Yaskawa INFORM job: A_ROOF_SIDE_0617_2_PAINT_49.JBI

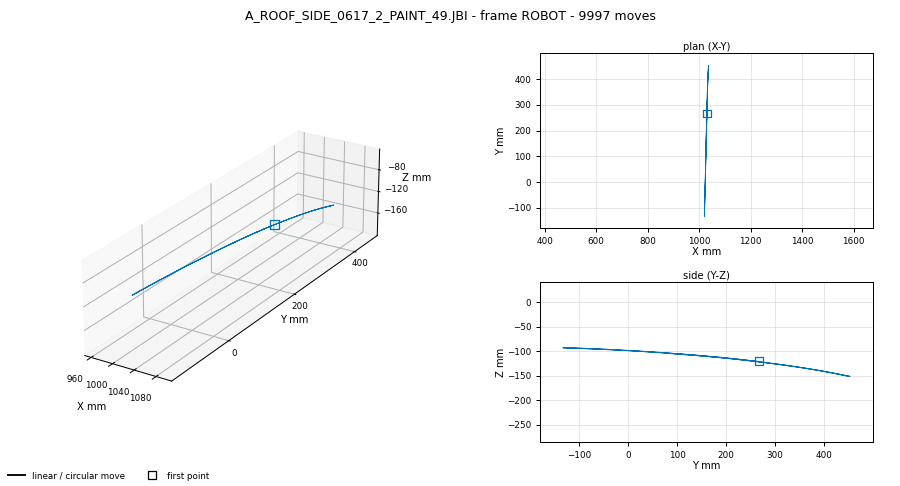
[picture p0: tool path of A_ROOF_SIDE_0617_2_PAINT_49.JBI in frame ROBOT, 9997 of 9997 moves have a stored position in this frame; points joined in program order, loops and branches not executed]
/JOB
//NAME A_ROOF_SIDE_0617_2_PAINT49
//POS
///NPOS 9997,0,0,0,0,0
///TOOL 1
///USER 0
///POSTYPE ROBOT
///RECTAN
///RCONF 1,0,0,0,0,0,0,0,0,0,0,0,0,0,0,0,0,0,0,0,0,0,0,0
C00000=1029.907,266.223,-120.891,170.566,45.689,158.767
C00001=1029.902,265.975,-120.861,170.562,45.690,158.767
C00002=1029.894,265.727,-120.831,170.558,45.691,158.767
C00003=1029.887,265.479,-120.801,170.555,45.691,158.766
C00004=1029.881,265.230,-120.772,170.551,45.692,158.766
C00005=1029.874,264.982,-120.741,170.547,45.693,158.766
C00006=1029.868,264.734,-120.711,170.544,45.694,158.766
C00007=1029.861,264.486,-120.681,170.539,45.695,158.766
C00008=1029.854,264.238,-120.651,170.536,45.696,158.765
C00009=1029.847,263.990,-120.622,170.532,45.697,158.765
C00010=1029.837,263.620,-120.577,170.527,45.697,158.765
C00011=1029.828,263.250,-120.532,170.521,45.699,158.764
C00012=1029.817,262.880,-120.488,170.516,45.700,158.764
C00013=1029.807,262.510,-120.443,170.511,45.701,158.764
C00014=1029.802,262.262,-120.413,170.507,45.702,158.764
C00015=1029.795,262.013,-120.383,170.503,45.703,158.763
C00016=1029.788,261.765,-120.354,170.500,45.704,158.763
C00017=1029.781,261.517,-120.324,170.496,45.705,158.763
C00018=1029.775,261.270,-120.294,170.493,45.705,158.763
C00019=1029.768,261.020,-120.264,170.489,45.706,158.763
C00020=1029.761,260.773,-120.235,170.486,45.708,158.763
C00021=1029.754,260.524,-120.205,170.482,45.709,158.762
C00022=1029.748,260.277,-120.176,170.478,45.710,158.762
C00023=1029.741,260.028,-120.146,170.475,45.710,158.762
C00024=1029.734,259.781,-120.117,170.471,45.711,158.762
C00025=1029.727,259.532,-120.088,170.468,45.713,158.762
C00026=1029.720,259.285,-120.058,170.464,45.714,158.761
C00027=1029.713,259.036,-120.029,170.460,45.715,158.761
C00028=1029.707,258.788,-120.000,170.457,45.715,158.761
C00029=1029.700,258.539,-119.969,170.453,45.717,158.761
C00030=1029.694,258.291,-119.940,170.450,45.718,158.761
C00031=1029.686,258.043,-119.912,170.446,45.719,158.761
C00032=1029.680,257.795,-119.882,170.442,45.720,158.760
C00033=1029.673,257.546,-119.852,170.439,45.721,158.760
C00034=1029.666,257.298,-119.823,170.435,45.722,158.760
C00035=1029.659,257.050,-119.793,170.432,45.723,158.760
C00036=1029.652,256.802,-119.765,170.428,45.724,158.760
C00037=1029.645,256.553,-119.735,170.425,45.725,158.760
C00038=1029.639,256.306,-119.706,170.421,45.726,158.760
C00039=1029.633,256.058,-119.677,170.417,45.727,158.759
C00040=1029.626,255.809,-119.647,170.414,45.728,158.759
C00041=1029.619,255.561,-119.619,170.410,45.729,158.759
C00042=1029.612,255.313,-119.589,170.407,45.730,158.759
C00043=1029.605,255.065,-119.560,170.403,45.731,158.759
C00044=1029.599,254.817,-119.531,170.401,45.732,158.759
C00045=1029.592,254.568,-119.501,170.397,45.733,158.758
C00046=1029.585,254.321,-119.472,170.393,45.734,158.758
C00047=1029.579,254.072,-119.443,170.390,45.735,158.758
C00048=1029.572,253.824,-119.414,170.387,45.736,158.758
C00049=1029.566,253.575,-119.385,170.383,45.737,158.758
C00050=1029.559,253.327,-119.355,170.380,45.739,158.758
C00051=1029.552,253.079,-119.327,170.376,45.739,158.758
C00052=1029.546,252.831,-119.298,170.372,45.740,158.757
C00053=1029.538,252.582,-119.267,170.369,45.742,158.757
C00054=1029.532,252.334,-119.238,170.365,45.743,158.757
C00055=1029.526,252.086,-119.209,170.362,45.743,158.757
C00056=1029.519,251.838,-119.181,170.358,45.745,158.757
C00057=1029.512,251.590,-119.152,170.355,45.746,158.757
C00058=1029.506,251.341,-119.123,170.351,45.747,158.757
C00059=1029.500,251.093,-119.093,170.348,45.748,158.756
C00060=1029.492,250.845,-119.065,170.344,45.749,158.756
C00061=1029.486,250.597,-119.036,170.342,45.750,158.756
C00062=1029.479,250.349,-119.007,170.337,45.751,158.756
C00063=1029.473,250.100,-118.978,170.335,45.753,158.756
C00064=1029.466,249.852,-118.948,170.332,45.753,158.756
C00065=1029.459,249.604,-118.920,170.328,45.754,158.756
C00066=1029.450,249.232,-118.876,170.323,45.756,158.755
C00067=1029.440,248.861,-118.833,170.318,45.758,158.755
C00068=1029.431,248.490,-118.789,170.312,45.760,158.755
C00069=1029.421,248.118,-118.746,170.307,45.761,158.755
C00070=1029.413,247.870,-118.717,170.304,45.762,158.755
C00071=1029.407,247.622,-118.688,170.300,45.764,158.755
C00072=1029.401,247.373,-118.660,170.297,45.764,158.754
C00073=1029.395,247.125,-118.631,170.295,45.766,158.754
C00074=1029.389,246.877,-118.602,170.291,45.767,158.754
C00075=1029.381,246.628,-118.573,170.288,45.768,158.754
C00076=1029.375,246.380,-118.544,170.284,45.769,158.754
C00077=1029.369,246.132,-118.515,170.281,45.770,158.754
C00078=1029.362,245.884,-118.486,170.277,45.771,158.754
C00079=1029.356,245.635,-118.458,170.274,45.773,158.754
C00080=1029.349,245.387,-118.429,170.271,45.774,158.753
C00081=1029.343,245.139,-118.400,170.267,45.774,158.753
C00082=1029.336,244.890,-118.371,170.264,45.776,158.753
C00083=1029.329,244.642,-118.342,170.260,45.777,158.753
C00084=1029.323,244.394,-118.314,170.258,45.778,158.753
C00085=1029.317,244.145,-118.285,170.254,45.780,158.753
C00086=1029.310,243.898,-118.256,170.251,45.780,158.753
C00087=1029.304,243.649,-118.228,170.248,45.782,158.753
C00088=1029.297,243.401,-118.200,170.244,45.783,158.752
C00089=1029.291,243.153,-118.170,170.241,45.784,158.752
C00090=1029.284,242.904,-118.142,170.237,45.786,158.752
C00091=1029.277,242.656,-118.113,170.234,45.786,158.752
C00092=1029.271,242.407,-118.086,170.231,45.788,158.752
C00093=1029.265,242.159,-118.057,170.228,45.789,158.752
C00094=1029.258,241.911,-118.028,170.224,45.790,158.752
C00095=1029.252,241.662,-118.000,170.221,45.792,158.752
C00096=1029.245,241.415,-117.971,170.218,45.793,158.752
C00097=1029.239,241.166,-117.943,170.214,45.794,158.752
C00098=1029.232,240.918,-117.915,170.211,45.795,158.752
C00099=1029.226,240.669,-117.886,170.208,45.797,158.752
C00100=1029.219,240.422,-117.858,170.205,45.798,158.751
C00101=1029.213,240.173,-117.829,170.202,45.799,158.751
C00102=1029.205,239.924,-117.801,170.198,45.801,158.751
C00103=1029.199,239.676,-117.773,170.195,45.802,158.751
C00104=1029.192,239.428,-117.744,170.191,45.803,158.751
C00105=1029.185,239.180,-117.717,170.188,45.804,158.751
C00106=1029.179,238.931,-117.688,170.185,45.806,158.751
C00107=1029.172,238.683,-117.660,170.182,45.807,158.751
C00108=1029.165,238.435,-117.632,170.178,45.809,158.751
C00109=1029.159,238.186,-117.605,170.175,45.810,158.751
C00110=1029.152,237.938,-117.575,170.172,45.811,158.751
C00111=1029.146,237.689,-117.548,170.169,45.813,158.751
C00112=1029.139,237.441,-117.520,170.166,45.814,158.751
C00113=1029.132,237.193,-117.492,170.162,45.816,158.751
C00114=1029.126,236.944,-117.463,170.159,45.817,158.751
C00115=1029.119,236.696,-117.436,170.157,45.818,158.751
C00116=1029.113,236.448,-117.408,170.153,45.820,158.750
C00117=1029.106,236.200,-117.379,170.150,45.821,158.750
C00118=1029.099,235.951,-117.352,170.146,45.822,158.750
C00119=1029.092,235.703,-117.324,170.143,45.824,158.750
C00120=1029.086,235.454,-117.296,170.139,45.825,158.750
C00121=1029.080,235.206,-117.268,170.137,45.827,158.750
C00122=1029.070,234.829,-117.225,170.132,45.829,158.750
C00123=1029.059,234.451,-117.182,170.127,45.831,158.750
C00124=1029.049,234.073,-117.140,170.123,45.833,158.750
C00125=1029.039,233.696,-117.098,170.117,45.836,158.750
C00126=1029.033,233.448,-117.070,170.114,45.837,158.750
C00127=1029.026,233.199,-117.042,170.111,45.838,158.750
C00128=1029.019,232.951,-117.014,170.107,45.839,158.750
C00129=1029.013,232.702,-116.987,170.105,45.841,158.750
C00130=1029.006,232.454,-116.959,170.102,45.842,158.750
C00131=1029.000,232.205,-116.931,170.098,45.844,158.750
C00132=1028.993,231.957,-116.903,170.095,45.845,158.750
C00133=1028.987,231.708,-116.875,170.092,45.847,158.749
C00134=1028.981,231.461,-116.848,170.089,45.848,158.749
C00135=1028.974,231.212,-116.820,170.086,45.849,158.749
C00136=1028.967,230.964,-116.792,170.082,45.851,158.749
C00137=1028.960,230.715,-116.765,170.080,45.852,158.749
C00138=1028.954,230.467,-116.737,170.077,45.854,158.749
C00139=1028.947,230.218,-116.709,170.073,45.855,158.749
C00140=1028.940,229.970,-116.681,170.070,45.857,158.749
C00141=1028.934,229.722,-116.654,170.066,45.858,158.749
C00142=1028.927,229.473,-116.626,170.064,45.860,158.749
C00143=1028.921,229.225,-116.599,170.061,45.861,158.749
C00144=1028.914,228.977,-116.571,170.057,45.863,158.749
C00145=1028.908,228.728,-116.543,170.055,45.865,158.749
C00146=1028.901,228.480,-116.515,170.052,45.866,158.749
C00147=1028.894,228.232,-116.488,170.048,45.868,158.749
C00148=1028.888,227.983,-116.461,170.045,45.869,158.749
C00149=1028.881,227.734,-116.433,170.043,45.870,158.749
C00150=1028.875,227.486,-116.406,170.039,45.872,158.749
C00151=1028.868,227.238,-116.378,170.036,45.873,158.749
C00152=1028.862,226.989,-116.350,170.032,45.875,158.749
C00153=1028.855,226.741,-116.324,170.030,45.876,158.749
C00154=1028.848,226.492,-116.296,170.027,45.878,158.749
C00155=1028.841,226.244,-116.268,170.023,45.880,158.749
C00156=1028.835,225.996,-116.241,170.021,45.881,158.749
C00157=1028.828,225.747,-116.214,170.018,45.883,158.749
C00158=1028.821,225.499,-116.187,170.014,45.885,158.749
C00159=1028.815,225.250,-116.159,170.012,45.886,158.749
C00160=1028.808,225.001,-116.132,170.009,45.888,158.749
C00161=1028.802,224.754,-116.105,170.005,45.889,158.749
C00162=1028.795,224.506,-116.078,170.002,45.891,158.749
C00163=1028.788,224.256,-116.050,169.999,45.893,158.749
C00164=1028.782,224.008,-116.023,169.996,45.894,158.749
C00165=1028.774,223.760,-115.996,169.993,45.896,158.749
C00166=1028.769,223.512,-115.969,169.989,45.897,158.749
C00167=1028.762,223.263,-115.941,169.987,45.899,158.749
C00168=1028.756,223.014,-115.914,169.984,45.901,158.749
C00169=1028.748,222.766,-115.887,169.980,45.902,158.749
C00170=1028.742,222.518,-115.860,169.978,45.904,158.749
C00171=1028.736,222.269,-115.833,169.975,45.906,158.749
C00172=1028.728,222.021,-115.806,169.971,45.907,158.749
C00173=1028.722,221.772,-115.779,169.969,45.909,158.749
C00174=1028.716,221.524,-115.751,169.966,45.910,158.749
C00175=1028.709,221.275,-115.724,169.962,45.912,158.749
C00176=1028.702,221.027,-115.697,169.960,45.914,158.749
C00177=1028.696,220.778,-115.670,169.957,45.915,158.749
C00178=1028.686,220.394,-115.628,169.952,45.918,158.749
C00179=1028.675,220.008,-115.586,169.948,45.920,158.749
C00180=1028.665,219.623,-115.544,169.942,45.923,158.749
C00181=1028.656,219.237,-115.502,169.938,45.925,158.749
C00182=1028.648,218.989,-115.475,169.935,45.927,158.749
C00183=1028.643,218.741,-115.448,169.932,45.929,158.749
C00184=1028.635,218.492,-115.422,169.929,45.930,158.749
C00185=1028.628,218.244,-115.394,169.926,45.932,158.749
C00186=1028.622,217.995,-115.367,169.923,45.934,158.749
C00187=1028.615,217.747,-115.341,169.920,45.936,158.749
C00188=1028.608,217.499,-115.314,169.917,45.937,158.749
C00189=1028.601,217.250,-115.287,169.915,45.939,158.750
C00190=1028.596,217.001,-115.261,169.911,45.941,158.750
C00191=1028.588,216.753,-115.233,169.908,45.943,158.750
C00192=1028.582,216.504,-115.206,169.906,45.944,158.750
C00193=1028.575,216.256,-115.180,169.902,45.946,158.750
C00194=1028.569,216.007,-115.153,169.899,45.948,158.750
C00195=1028.561,215.759,-115.126,169.897,45.949,158.750
C00196=1028.555,215.511,-115.100,169.893,45.952,158.750
C00197=1028.549,215.262,-115.073,169.890,45.953,158.750
C00198=1028.542,215.014,-115.047,169.888,45.955,158.750
C00199=1028.536,214.765,-115.020,169.884,45.957,158.750
C00200=1028.528,214.517,-114.993,169.882,45.959,158.750
C00201=1028.523,214.268,-114.966,169.879,45.960,158.750
C00202=1028.515,214.020,-114.940,169.876,45.962,158.750
C00203=1028.508,213.771,-114.913,169.873,45.964,158.750
C00204=1028.503,213.522,-114.887,169.870,45.966,158.750
C00205=1028.495,213.274,-114.860,169.867,45.967,158.750
C00206=1028.489,213.026,-114.833,169.864,45.969,158.750
C00207=1028.482,212.777,-114.807,169.861,45.971,158.750
C00208=1028.476,212.529,-114.780,169.859,45.973,158.750
C00209=1028.469,212.280,-114.754,169.856,45.974,158.750
C00210=1028.463,212.031,-114.727,169.852,45.976,158.751
C00211=1028.456,211.783,-114.700,169.850,45.978,158.750
C00212=1028.449,211.534,-114.674,169.847,45.980,158.751
C00213=1028.444,211.286,-114.647,169.843,45.981,158.751
C00214=1028.436,211.038,-114.620,169.841,45.983,158.751
C00215=1028.430,210.789,-114.594,169.838,45.985,158.751
C00216=1028.423,210.541,-114.567,169.836,45.987,158.751
C00217=1028.417,210.293,-114.541,169.832,45.988,158.751
C00218=1028.410,210.044,-114.515,169.829,45.990,158.751
C00219=1028.403,209.795,-114.488,169.827,45.993,158.751
C00220=1028.397,209.547,-114.462,169.823,45.994,158.751
C00221=1028.390,209.298,-114.435,169.821,45.996,158.751
C00222=1028.383,209.050,-114.409,169.818,45.998,158.751
C00223=1028.377,208.800,-114.383,169.815,46.000,158.751
C00224=1028.371,208.552,-114.357,169.812,46.002,158.751
C00225=1028.363,208.303,-114.330,169.809,46.003,158.751
C00226=1028.357,208.055,-114.304,169.807,46.005,158.751
C00227=1028.351,207.806,-114.277,169.803,46.008,158.752
C00228=1028.344,207.558,-114.251,169.801,46.010,158.752
C00229=1028.337,207.309,-114.225,169.798,46.011,158.752
C00230=1028.330,207.061,-114.199,169.795,46.013,158.752
C00231=1028.323,206.813,-114.172,169.792,46.015,158.752
C00232=1028.317,206.564,-114.147,169.789,46.017,158.752
C00233=1028.311,206.315,-114.120,169.787,46.019,158.752
C00234=1028.300,205.936,-114.080,169.782,46.022,158.752
C00235=1028.290,205.556,-114.040,169.778,46.024,158.752
C00236=1028.280,205.176,-114.001,169.774,46.027,158.752
C00237=1028.269,204.795,-113.961,169.769,46.031,158.753
C00238=1028.244,203.751,-113.857,169.396,45.927,158.689
C00239=1028.238,203.502,-113.832,169.392,45.930,158.689
C00240=1028.233,203.253,-113.808,169.388,45.932,158.689
C00241=1028.227,203.005,-113.783,169.384,45.936,158.690
C00242=1028.220,202.756,-113.759,169.380,45.938,158.690
C00243=1028.215,202.508,-113.734,169.376,45.941,158.690
C00244=1028.209,202.258,-113.709,169.372,45.943,158.690
C00245=1028.203,202.009,-113.684,169.369,45.946,158.690
C00246=1028.197,201.761,-113.659,169.365,45.949,158.690
C00247=1028.191,201.512,-113.635,169.361,45.952,158.690
C00248=1028.185,201.264,-113.611,169.357,45.954,158.690
C00249=1028.179,201.015,-113.586,169.354,45.957,158.691
C00250=1028.174,200.766,-113.562,169.349,45.960,158.691
C00251=1028.168,200.517,-113.537,169.346,45.963,158.691
C00252=1028.162,200.268,-113.512,169.342,45.965,158.691
C00253=1028.156,200.020,-113.488,169.338,45.968,158.691
C00254=1028.150,199.771,-113.463,169.335,45.971,158.691
C00255=1028.144,199.523,-113.440,169.331,45.974,158.692
C00256=1028.138,199.273,-113.415,169.327,45.976,158.692
C00257=1028.132,199.025,-113.391,169.323,45.980,158.692
C00258=1028.126,198.776,-113.367,169.320,45.982,158.692
C00259=1028.119,198.527,-113.343,169.315,45.985,158.692
C00260=1028.113,198.278,-113.319,169.312,45.988,158.692
C00261=1028.107,198.030,-113.294,169.308,45.991,158.692
C00262=1028.101,197.782,-113.270,169.304,45.994,158.693
C00263=1028.095,197.532,-113.245,169.301,45.996,158.693
C00264=1028.089,197.284,-113.222,169.297,45.999,158.693
C00265=1028.083,197.035,-113.197,169.293,46.002,158.693
C00266=1028.077,196.786,-113.173,169.289,46.006,158.693
C00267=1028.071,196.537,-113.149,169.286,46.008,158.693
C00268=1028.065,196.289,-113.125,169.282,46.011,158.694
C00269=1028.059,196.040,-113.101,169.278,46.014,158.694
C00270=1028.053,195.791,-113.077,169.275,46.017,158.694
C00271=1028.047,195.542,-113.053,169.271,46.020,158.694
C00272=1028.041,195.294,-113.029,169.267,46.022,158.694
C00273=1028.035,195.045,-113.005,169.264,46.025,158.695
C00274=1028.030,194.795,-112.981,169.260,46.028,158.695
C00275=1028.024,194.547,-112.957,169.256,46.031,158.695
C00276=1028.018,194.298,-112.933,169.252,46.035,158.695
C00277=1028.012,194.050,-112.909,169.249,46.037,158.695
C00278=1028.006,193.800,-112.885,169.245,46.040,158.695
C00279=1028.000,193.552,-112.861,169.241,46.043,158.696
C00280=1027.993,193.303,-112.837,169.238,46.046,158.696
C00281=1027.988,193.055,-112.813,169.235,46.049,158.696
C00282=1027.982,192.806,-112.789,169.230,46.051,158.696
C00283=1027.976,192.556,-112.765,169.227,46.054,158.696
C00284=1027.970,192.308,-112.741,169.224,46.057,158.697
C00285=1027.965,192.059,-112.717,169.219,46.060,158.697
C00286=1027.958,191.810,-112.693,169.216,46.063,158.697
C00287=1027.952,191.562,-112.669,169.213,46.066,158.697
C00288=1027.947,191.312,-112.645,169.208,46.069,158.697
C00289=1027.941,191.064,-112.622,169.205,46.072,158.697
C00290=1027.935,190.815,-112.598,169.202,46.075,158.698
C00291=1027.929,190.566,-112.574,169.198,46.078,158.698
C00292=1027.924,190.317,-112.550,169.194,46.081,158.698
C00293=1027.918,190.069,-112.526,169.191,46.083,158.698
C00294=1027.912,189.821,-112.503,169.187,46.086,158.698
C00295=1027.906,189.571,-112.478,169.183,46.089,158.699
C00296=1027.900,189.323,-112.455,169.180,46.092,158.699
C00297=1027.895,189.074,-112.431,169.177,46.095,158.699
C00298=1027.888,188.825,-112.407,169.173,46.098,158.699
C00299=1027.882,188.542,-112.379,169.169,46.101,158.699
C00300=1027.875,188.259,-112.353,169.165,46.104,158.700
C00301=1027.869,187.976,-112.326,169.161,46.108,158.700
C00302=1027.862,187.693,-112.299,169.157,46.111,158.700
C00303=1027.857,187.444,-112.275,169.154,46.114,158.700
C00304=1027.851,187.196,-112.252,169.149,46.117,158.700
C00305=1027.844,186.947,-112.228,169.146,46.120,158.701
C00306=1027.839,186.697,-112.204,169.143,46.123,158.701
C00307=1027.833,186.449,-112.181,169.140,46.126,158.701
C00308=1027.828,186.200,-112.157,169.135,46.129,158.701
C00309=1027.822,185.952,-112.133,169.132,46.132,158.701
C00310=1027.815,185.703,-112.109,169.129,46.135,158.702
C00311=1027.810,185.453,-112.086,169.125,46.137,158.702
C00312=1027.804,185.205,-112.062,169.122,46.140,158.702
C00313=1027.799,184.956,-112.039,169.118,46.143,158.702
C00314=1027.793,184.708,-112.015,169.115,46.146,158.702
C00315=1027.787,184.459,-111.992,169.111,46.149,158.703
C00316=1027.782,184.209,-111.967,169.108,46.152,158.703
C00317=1027.776,183.961,-111.944,169.105,46.155,158.703
C00318=1027.771,183.712,-111.920,169.101,46.158,158.703
C00319=1027.765,183.463,-111.897,169.097,46.161,158.703
C00320=1027.759,183.215,-111.874,169.094,46.164,158.703
C00321=1027.753,182.965,-111.850,169.091,46.166,158.704
C00322=1027.747,182.716,-111.827,169.087,46.169,158.704
C00323=1027.741,182.468,-111.803,169.083,46.173,158.704
C00324=1027.736,182.219,-111.780,169.080,46.176,158.705
C00325=1027.729,181.969,-111.757,169.077,46.179,158.705
C00326=1027.723,181.721,-111.734,169.073,46.182,158.705
C00327=1027.717,181.472,-111.711,169.070,46.185,158.705
C00328=1027.711,181.223,-111.689,169.066,46.188,158.705
C00329=1027.705,180.975,-111.665,169.063,46.192,158.706
C00330=1027.700,180.726,-111.642,169.059,46.195,158.706
C00331=1027.693,180.476,-111.619,169.056,46.198,158.706
C00332=1027.687,180.227,-111.596,169.053,46.201,158.706
C00333=1027.681,179.979,-111.573,169.048,46.204,158.707
C00334=1027.675,179.730,-111.550,169.045,46.208,158.707
C00335=1027.669,179.481,-111.528,169.042,46.211,158.707
C00336=1027.663,179.232,-111.505,169.039,46.214,158.707
C00337=1027.657,178.983,-111.481,169.035,46.217,158.708
C00338=1027.651,178.734,-111.458,169.032,46.221,158.708
C00339=1027.645,178.485,-111.435,169.029,46.224,158.708
C00340=1027.639,178.237,-111.413,169.025,46.227,158.708
C00341=1027.633,177.988,-111.390,169.022,46.230,158.709
C00342=1027.627,177.739,-111.367,169.018,46.233,158.709
C00343=1027.621,177.490,-111.344,169.015,46.236,158.709
C00344=1027.615,177.242,-111.322,169.012,46.239,158.709
C00345=1027.609,176.992,-111.298,169.009,46.242,158.710
C00346=1027.603,176.743,-111.275,169.004,46.245,158.710
C00347=1027.597,176.494,-111.252,169.001,46.249,158.710
C00348=1027.591,176.246,-111.230,168.998,46.252,158.710
C00349=1027.585,175.997,-111.207,168.995,46.255,158.711
C00350=1027.579,175.748,-111.184,168.992,46.258,158.711
C00351=1027.573,175.499,-111.161,168.988,46.262,158.711
C00352=1027.567,175.250,-111.139,168.984,46.265,158.711
C00353=1027.561,175.001,-111.116,168.981,46.268,158.712
C00354=1027.556,174.753,-111.093,168.978,46.271,158.712
C00355=1027.550,174.504,-111.070,168.975,46.274,158.712
C00356=1027.544,174.254,-111.048,168.972,46.277,158.712
C00357=1027.538,174.006,-111.025,168.968,46.281,158.713
C00358=1027.532,173.757,-111.003,168.964,46.284,158.713
C00359=1027.526,173.508,-110.980,168.961,46.287,158.713
C00360=1027.520,173.259,-110.957,168.958,46.290,158.714
C00361=1027.514,173.010,-110.934,168.955,46.293,158.714
C00362=1027.509,172.761,-110.911,168.952,46.296,158.714
C00363=1027.502,172.478,-110.886,168.948,46.300,158.714
C00364=1027.495,172.194,-110.860,168.944,46.304,158.715
C00365=1027.488,171.911,-110.834,168.940,46.308,158.715
C00366=1027.482,171.627,-110.808,168.937,46.311,158.715
C00367=1027.476,171.378,-110.786,168.934,46.314,158.716
C00368=1027.470,171.129,-110.763,168.930,46.317,158.716
C00369=1027.464,170.881,-110.740,168.926,46.320,158.716
C00370=1027.459,170.631,-110.718,168.923,46.323,158.716
C00371=1027.452,170.382,-110.695,168.920,46.327,158.717
C00372=1027.447,170.134,-110.673,168.917,46.330,158.717
C00373=1027.441,169.885,-110.650,168.914,46.333,158.717
C00374=1027.435,169.635,-110.627,168.910,46.336,158.717
C00375=1027.430,169.387,-110.605,168.907,46.340,158.718
C00376=1027.424,169.138,-110.582,168.904,46.343,158.718
C00377=1027.418,168.889,-110.559,168.901,46.346,158.718
C00378=1027.412,168.640,-110.538,168.898,46.349,158.718
C00379=1027.406,168.391,-110.515,168.894,46.352,158.719
C00380=1027.401,168.142,-110.492,168.891,46.355,158.719
C00381=1027.395,167.893,-110.470,168.887,46.358,158.719
C00382=1027.389,167.644,-110.447,168.884,46.362,158.719
C00383=1027.383,167.396,-110.425,168.881,46.365,158.720
C00384=1027.378,167.147,-110.403,168.878,46.368,158.720
C00385=1027.372,166.898,-110.380,168.875,46.371,158.720
C00386=1027.366,166.649,-110.357,168.872,46.375,158.720
C00387=1027.360,166.400,-110.335,168.869,46.378,158.721
C00388=1027.355,166.151,-110.312,168.865,46.381,158.721
C00389=1027.349,165.902,-110.291,168.862,46.384,158.721
C00390=1027.343,165.653,-110.268,168.859,46.387,158.722
C00391=1027.338,165.404,-110.245,168.856,46.390,158.722
C00392=1027.332,165.155,-110.223,168.853,46.393,158.722
C00393=1027.326,164.906,-110.200,168.850,46.397,158.722
C00394=1027.320,164.657,-110.178,168.847,46.400,158.723
C00395=1027.315,164.409,-110.156,168.843,46.403,158.723
C00396=1027.309,164.160,-110.133,168.840,46.406,158.723
C00397=1027.303,163.911,-110.111,168.837,46.409,158.723
C00398=1027.298,163.662,-110.088,168.834,46.412,158.724
C00399=1027.292,163.413,-110.067,168.831,46.415,158.724
C00400=1027.286,163.164,-110.044,168.827,46.418,158.724
C00401=1027.281,162.915,-110.022,168.825,46.422,158.724
C00402=1027.275,162.666,-109.999,168.821,46.425,158.725
C00403=1027.270,162.417,-109.977,168.818,46.428,158.725
C00404=1027.264,162.168,-109.954,168.815,46.432,158.725
C00405=1027.258,161.919,-109.932,168.812,46.435,158.726
C00406=1027.252,161.670,-109.910,168.809,46.438,158.726
C00407=1027.247,161.422,-109.888,168.805,46.441,158.726
C00408=1027.242,161.172,-109.866,168.803,46.444,158.726
C00409=1027.235,160.923,-109.843,168.799,46.447,158.727
C00410=1027.230,160.675,-109.821,168.796,46.450,158.727
C00411=1027.225,160.426,-109.799,168.793,46.453,158.727
C00412=1027.219,160.176,-109.776,168.790,46.457,158.727
C00413=1027.213,159.928,-109.754,168.787,46.460,158.728
C00414=1027.208,159.679,-109.732,168.784,46.463,158.728
C00415=1027.203,159.429,-109.710,168.781,46.467,158.728
C00416=1027.196,159.181,-109.688,168.777,46.470,158.728
C00417=1027.191,158.932,-109.666,168.774,46.473,158.729
C00418=1027.184,158.683,-109.645,168.771,46.476,158.729
C00419=1027.179,158.433,-109.622,168.768,46.480,158.729
C00420=1027.173,158.184,-109.601,168.765,46.483,158.730
C00421=1027.167,157.936,-109.579,168.762,46.486,158.730
C00422=1027.161,157.687,-109.557,168.759,46.489,158.730
C00423=1027.155,157.438,-109.535,168.756,46.493,158.731
C00424=1027.150,157.189,-109.514,168.753,46.496,158.731
C00425=1027.144,156.940,-109.492,168.750,46.500,158.731
C00426=1027.137,156.691,-109.470,168.747,46.503,158.731
C00427=1027.131,156.407,-109.445,168.743,46.507,158.732
C00428=1027.124,156.124,-109.420,168.740,46.510,158.732
C00429=1027.118,155.839,-109.396,168.736,46.514,158.732
C00430=1027.111,155.556,-109.371,168.733,46.518,158.733
C00431=1027.106,155.306,-109.349,168.730,46.522,158.733
C00432=1027.100,155.057,-109.327,168.727,46.525,158.733
C00433=1027.094,154.809,-109.306,168.724,46.528,158.734
C00434=1027.088,154.559,-109.284,168.721,46.531,158.734
C00435=1027.082,154.310,-109.262,168.718,46.535,158.734
C00436=1027.077,154.061,-109.241,168.714,46.538,158.735
C00437=1027.071,153.812,-109.219,168.711,46.542,158.735
C00438=1027.065,153.563,-109.197,168.708,46.545,158.735
C00439=1027.059,153.314,-109.176,168.705,46.548,158.736
C00440=1027.054,153.065,-109.154,168.702,46.551,158.736
C00441=1027.047,152.816,-109.132,168.699,46.555,158.736
C00442=1027.042,152.567,-109.111,168.696,46.558,158.736
C00443=1027.036,152.318,-109.089,168.693,46.562,158.737
C00444=1027.030,152.069,-109.068,168.690,46.565,158.737
C00445=1027.024,151.820,-109.047,168.687,46.568,158.737
C00446=1027.018,151.571,-109.025,168.684,46.572,158.738
C00447=1027.012,151.323,-109.004,168.681,46.575,158.738
C00448=1027.006,151.073,-108.982,168.678,46.579,158.738
C00449=1027.000,150.825,-108.961,168.675,46.582,158.739
C00450=1026.994,150.576,-108.939,168.672,46.585,158.739
C00451=1026.989,150.325,-108.918,168.668,46.588,158.739
C00452=1026.984,150.077,-108.896,168.666,46.592,158.740
C00453=1026.977,149.828,-108.875,168.663,46.596,158.740
C00454=1026.972,149.579,-108.853,168.659,46.599,158.740
C00455=1026.966,149.330,-108.832,168.657,46.602,158.741
C00456=1026.960,149.082,-108.810,168.654,46.605,158.741
C00457=1026.954,148.832,-108.789,168.651,46.609,158.741
C00458=1026.948,148.583,-108.768,168.648,46.612,158.741
C00459=1026.943,148.334,-108.747,168.645,46.615,158.742
C00460=1026.936,148.085,-108.725,168.642,46.619,158.742
C00461=1026.931,147.836,-108.704,168.639,46.622,158.742
C00462=1026.925,147.587,-108.682,168.636,46.626,158.743
C00463=1026.919,147.338,-108.662,168.633,46.629,158.743
C00464=1026.913,147.089,-108.640,168.630,46.632,158.743
C00465=1026.908,146.840,-108.619,168.627,46.636,158.744
C00466=1026.902,146.590,-108.598,168.624,46.639,158.744
C00467=1026.896,146.342,-108.576,168.621,46.643,158.744
C00468=1026.890,146.093,-108.555,168.618,46.646,158.745
C00469=1026.885,145.844,-108.534,168.616,46.649,158.745
C00470=1026.879,145.594,-108.513,168.613,46.653,158.745
C00471=1026.872,145.346,-108.492,168.610,46.657,158.746
C00472=1026.867,145.096,-108.471,168.607,46.660,158.746
C00473=1026.861,144.848,-108.450,168.604,46.663,158.746
C00474=1026.855,144.599,-108.428,168.601,46.667,158.747
C00475=1026.850,144.350,-108.408,168.598,46.670,158.747
C00476=1026.843,144.101,-108.387,168.595,46.674,158.747
C00477=1026.837,143.852,-108.366,168.592,46.677,158.748
C00478=1026.831,143.602,-108.344,168.589,46.680,158.748
C00479=1026.826,143.354,-108.323,168.586,46.684,158.748
C00480=1026.820,143.104,-108.302,168.583,46.688,158.749
C00481=1026.814,142.856,-108.281,168.580,46.691,158.749
C00482=1026.808,142.606,-108.261,168.577,46.694,158.749
C00483=1026.802,142.358,-108.239,168.575,46.698,158.750
C00484=1026.796,142.108,-108.218,168.572,46.701,158.750
C00485=1026.791,141.859,-108.197,168.569,46.705,158.750
C00486=1026.785,141.609,-108.176,168.566,46.708,158.751
C00487=1026.779,141.361,-108.156,168.563,46.711,158.751
C00488=1026.773,141.112,-108.135,168.560,46.715,158.751
C00489=1026.767,140.863,-108.113,168.557,46.719,158.752
C00490=1026.762,140.614,-108.093,168.553,46.722,158.752
C00491=1026.755,140.330,-108.069,168.551,46.726,158.752
C00492=1026.748,140.046,-108.045,168.547,46.730,158.753
C00493=1026.742,139.762,-108.021,168.544,46.734,158.753
C00494=1026.735,139.477,-107.997,168.541,46.737,158.753
C00495=1026.729,139.228,-107.976,168.538,46.741,158.754
C00496=1026.724,138.979,-107.955,168.535,46.745,158.754
C00497=1026.718,138.730,-107.935,168.532,46.748,158.754
C00498=1026.712,138.481,-107.914,168.529,46.752,158.755
C00499=1026.706,138.231,-107.893,168.526,46.755,158.755
C00500=1026.700,137.983,-107.872,168.523,46.758,158.755
C00501=1026.694,137.733,-107.852,168.521,46.762,158.756
C00502=1026.689,137.484,-107.831,168.518,46.765,158.756
C00503=1026.682,137.235,-107.810,168.515,46.769,158.757
C00504=1026.677,136.986,-107.789,168.512,46.772,158.757
C00505=1026.670,136.737,-107.769,168.509,46.776,158.757
C00506=1026.665,136.488,-107.748,168.506,46.780,158.758
C00507=1026.660,136.239,-107.727,168.503,46.783,158.758
C00508=1026.653,135.990,-107.707,168.500,46.786,158.758
C00509=1026.647,135.741,-107.686,168.497,46.790,158.758
C00510=1026.641,135.492,-107.666,168.495,46.793,158.759
C00511=1026.635,135.242,-107.645,168.492,46.797,158.759
C00512=1026.629,134.994,-107.625,168.489,46.800,158.760
C00513=1026.624,134.744,-107.604,168.486,46.804,158.760
C00514=1026.618,134.495,-107.583,168.483,46.808,158.760
C00515=1026.612,134.246,-107.563,168.480,46.811,158.761
C00516=1026.607,133.997,-107.542,168.477,46.814,158.761
C00517=1026.600,133.748,-107.522,168.475,46.818,158.761
C00518=1026.595,133.499,-107.501,168.472,46.821,158.762
C00519=1026.589,133.251,-107.481,168.469,46.825,158.762
C00520=1026.583,133.001,-107.460,168.466,46.828,158.762
C00521=1026.577,132.752,-107.440,168.463,46.832,158.763
C00522=1026.572,132.503,-107.419,168.460,46.836,158.763
C00523=1026.565,132.253,-107.399,168.458,46.839,158.763
C00524=1026.560,132.004,-107.378,168.456,46.843,158.764
C00525=1026.553,131.756,-107.358,168.452,46.846,158.764
C00526=1026.548,131.507,-107.337,168.450,46.849,158.764
C00527=1026.542,131.257,-107.317,168.447,46.853,158.765
C00528=1026.536,131.008,-107.296,168.443,46.856,158.765
C00529=1026.530,130.759,-107.276,168.442,46.860,158.765
C00530=1026.525,130.510,-107.256,168.439,46.863,158.766
C00531=1026.518,130.261,-107.235,168.436,46.867,158.766
C00532=1026.513,130.012,-107.215,168.433,46.871,158.767
C00533=1026.507,129.763,-107.195,168.430,46.874,158.767
C00534=1026.501,129.513,-107.174,168.427,46.878,158.767
C00535=1026.495,129.264,-107.155,168.424,46.881,158.767
C00536=1026.489,129.015,-107.134,168.421,46.885,158.768
C00537=1026.483,128.767,-107.114,168.419,46.888,158.768
C00538=1026.477,128.517,-107.094,168.416,46.892,158.769
C00539=1026.471,128.268,-107.074,168.413,46.896,158.769
C00540=1026.465,128.019,-107.054,168.410,46.900,158.769
C00541=1026.459,127.769,-107.034,168.407,46.903,158.770
C00542=1026.453,127.520,-107.014,168.404,46.907,158.770
C00543=1026.447,127.271,-106.994,168.402,46.911,158.771
C00544=1026.441,127.022,-106.974,168.399,46.914,158.771
C00545=1026.435,126.773,-106.953,168.397,46.918,158.771
C00546=1026.429,126.524,-106.933,168.394,46.921,158.772
C00547=1026.423,126.275,-106.913,168.391,46.925,158.772
C00548=1026.417,126.026,-106.893,168.388,46.928,158.772
C00549=1026.412,125.777,-106.874,168.385,46.932,158.773
C00550=1026.405,125.527,-106.853,168.382,46.936,158.773
C00551=1026.399,125.278,-106.833,168.380,46.939,158.773
C00552=1026.394,125.029,-106.813,168.377,46.943,158.774
C00553=1026.388,124.781,-106.793,168.374,46.947,158.774
C00554=1026.382,124.531,-106.774,168.371,46.950,158.775
C00555=1026.375,124.247,-106.751,168.368,46.954,158.775
C00556=1026.369,123.962,-106.728,168.364,46.958,158.775
C00557=1026.362,123.678,-106.705,168.362,46.962,158.776
C00558=1026.354,123.393,-106.682,168.359,46.966,158.776
C00559=1026.349,123.144,-106.662,168.356,46.970,158.777
C00560=1026.343,122.895,-106.642,168.353,46.974,158.777
C00561=1026.337,122.647,-106.622,168.350,46.977,158.777
C00562=1026.331,122.397,-106.603,168.347,46.981,158.778
C00563=1026.325,122.148,-106.583,168.345,46.985,158.778
C00564=1026.319,121.900,-106.563,168.342,46.988,158.778
C00565=1026.314,121.650,-106.542,168.339,46.991,158.779
C00566=1026.308,121.400,-106.522,168.336,46.995,158.779
C00567=1026.302,121.151,-106.502,168.334,46.999,158.779
C00568=1026.296,120.903,-106.483,168.332,47.002,158.780
C00569=1026.290,120.653,-106.463,168.329,47.006,158.780
C00570=1026.284,120.404,-106.443,168.326,47.010,158.781
C00571=1026.279,120.155,-106.423,168.323,47.013,158.781
C00572=1026.273,119.906,-106.404,168.320,47.016,158.781
C00573=1026.267,119.656,-106.383,168.318,47.020,158.782
C00574=1026.261,119.408,-106.363,168.315,47.024,158.782
C00575=1026.255,119.158,-106.344,168.312,47.027,158.782
C00576=1026.249,118.909,-106.324,168.309,47.031,158.783
C00577=1026.244,118.660,-106.303,168.307,47.034,158.783
C00578=1026.238,118.411,-106.284,168.304,47.038,158.783
C00579=1026.232,118.162,-106.264,168.301,47.041,158.784
C00580=1026.226,117.913,-106.244,168.298,47.045,158.784
C00581=1026.220,117.664,-106.225,168.296,47.049,158.785
C00582=1026.214,117.415,-106.205,168.293,47.052,158.785
C00583=1026.209,117.165,-106.186,168.290,47.055,158.785
C00584=1026.203,116.916,-106.165,168.288,47.059,158.785
C00585=1026.197,116.667,-106.145,168.286,47.063,158.786
C00586=1026.192,116.418,-106.126,168.283,47.066,158.786
C00587=1026.186,116.169,-106.106,168.280,47.069,158.786
C00588=1026.180,115.920,-106.087,168.277,47.073,158.787
C00589=1026.174,115.670,-106.067,168.275,47.077,158.787
C00590=1026.169,115.421,-106.047,168.272,47.080,158.788
C00591=1026.163,115.172,-106.027,168.269,47.084,158.788
C00592=1026.157,114.922,-106.008,168.266,47.087,158.788
C00593=1026.151,114.673,-105.988,168.264,47.091,158.789
C00594=1026.145,114.425,-105.968,168.261,47.094,158.789
C00595=1026.139,114.175,-105.948,168.258,47.098,158.789
C00596=1026.133,113.926,-105.928,168.256,47.102,158.790
C00597=1026.128,113.677,-105.909,168.253,47.105,158.790
C00598=1026.122,113.428,-105.889,168.250,47.108,158.790
C00599=1026.117,113.178,-105.869,168.247,47.112,158.791
C00600=1026.111,112.929,-105.850,168.245,47.116,158.791
C00601=1026.105,112.680,-105.830,168.242,47.119,158.791
C00602=1026.099,112.431,-105.811,168.239,47.122,158.792
C00603=1026.093,112.182,-105.791,168.236,47.126,158.792
C00604=1026.088,111.932,-105.772,168.235,47.130,158.793
C00605=1026.082,111.683,-105.753,168.232,47.133,158.793
C00606=1026.075,111.435,-105.733,168.229,47.137,158.793
C00607=1026.069,111.185,-105.714,168.226,47.141,158.794
C00608=1026.064,110.936,-105.695,168.224,47.144,158.794
C00609=1026.058,110.687,-105.675,168.221,47.148,158.794
C00610=1026.052,110.437,-105.655,168.218,47.152,158.795
C00611=1026.046,110.188,-105.636,168.215,47.156,158.795
C00612=1026.041,109.939,-105.617,168.213,47.159,158.796
C00613=1026.035,109.691,-105.598,168.211,47.163,158.796
C00614=1026.029,109.441,-105.579,168.208,47.167,158.796
C00615=1026.023,109.192,-105.559,168.205,47.170,158.797
C00616=1026.017,108.943,-105.541,168.203,47.174,158.797
C00617=1026.011,108.694,-105.521,168.200,47.177,158.797
C00618=1026.005,108.445,-105.502,168.197,47.181,158.798
C00619=1025.998,108.160,-105.480,168.194,47.185,158.798
C00620=1025.991,107.876,-105.459,168.191,47.190,158.799
C00621=1025.984,107.591,-105.437,168.188,47.193,158.799
C00622=1025.977,107.306,-105.414,168.185,47.198,158.800
C00623=1025.972,107.058,-105.395,168.182,47.202,158.800
C00624=1025.966,106.808,-105.376,168.179,47.205,158.800
C00625=1025.960,106.559,-105.357,168.178,47.209,158.801
C00626=1025.954,106.310,-105.338,168.175,47.213,158.801
C00627=1025.948,106.060,-105.319,168.171,47.216,158.801
C00628=1025.942,105.812,-105.299,168.169,47.219,158.802
C00629=1025.936,105.562,-105.280,168.166,47.223,158.802
C00630=1025.930,105.313,-105.261,168.164,47.227,158.803
C00631=1025.924,105.064,-105.242,168.161,47.230,158.803
C00632=1025.918,104.814,-105.223,168.158,47.234,158.803
C00633=1025.912,104.565,-105.204,168.156,47.238,158.804
C00634=1025.907,104.316,-105.185,168.153,47.241,158.804
C00635=1025.901,104.067,-105.166,168.150,47.245,158.804
C00636=1025.895,103.818,-105.148,168.148,47.249,158.805
C00637=1025.889,103.568,-105.128,168.146,47.252,158.805
C00638=1025.883,103.319,-105.109,168.143,47.256,158.806
C00639=1025.877,103.070,-105.090,168.140,47.260,158.806
C00640=1025.871,102.820,-105.071,168.137,47.264,158.806
C00641=1025.865,102.572,-105.051,168.135,47.267,158.807
C00642=1025.860,102.323,-105.033,168.132,47.270,158.807
C00643=1025.854,102.074,-105.014,168.129,47.274,158.807
C00644=1025.848,101.824,-104.994,168.127,47.278,158.808
C00645=1025.842,101.575,-104.976,168.124,47.281,158.808
C00646=1025.836,101.326,-104.957,168.121,47.285,158.808
C00647=1025.830,101.076,-104.937,168.119,47.289,158.809
C00648=1025.825,100.828,-104.919,168.117,47.292,158.809
C00649=1025.819,100.578,-104.900,168.114,47.296,158.810
C00650=1025.813,100.329,-104.881,168.111,47.300,158.810
C00651=1025.807,100.079,-104.863,168.109,47.303,158.810
C00652=1025.801,99.830,-104.843,168.106,47.306,158.811
C00653=1025.796,99.580,-104.824,168.103,47.310,158.811
C00654=1025.790,99.332,-104.806,168.100,47.314,158.811
C00655=1025.783,99.083,-104.787,168.098,47.317,158.812
C00656=1025.778,98.833,-104.768,168.095,47.321,158.812
C00657=1025.771,98.584,-104.749,168.093,47.325,158.812
C00658=1025.766,98.334,-104.731,168.090,47.329,158.813
C00659=1025.759,98.085,-104.712,168.088,47.333,158.813
C00660=1025.754,97.837,-104.694,168.085,47.337,158.814
C00661=1025.748,97.587,-104.675,168.082,47.341,158.814
C00662=1025.742,97.338,-104.656,168.079,47.344,158.815
C00663=1025.736,97.088,-104.637,168.078,47.348,158.815
C00664=1025.730,96.839,-104.619,168.075,47.352,158.815
C00665=1025.724,96.591,-104.600,168.072,47.355,158.816
C00666=1025.718,96.341,-104.581,168.070,47.359,158.816
C00667=1025.712,96.092,-104.563,168.067,47.363,158.816
C00668=1025.706,95.842,-104.545,168.064,47.366,158.817
C00669=1025.700,95.593,-104.525,168.061,47.370,158.817
C00670=1025.694,95.344,-104.507,168.060,47.374,158.818
C00671=1025.688,95.095,-104.488,168.057,47.377,158.818
C00672=1025.682,94.845,-104.470,168.054,47.381,158.818
C00673=1025.676,94.596,-104.451,168.051,47.385,158.819
C00674=1025.671,94.347,-104.432,168.049,47.388,158.819
C00675=1025.665,94.098,-104.415,168.046,47.392,158.820
C00676=1025.658,93.848,-104.396,168.043,47.396,158.820
C00677=1025.653,93.599,-104.377,168.041,47.399,158.820
C00678=1025.647,93.350,-104.359,168.038,47.403,158.821
C00679=1025.641,93.101,-104.340,168.035,47.406,158.821
C00680=1025.635,92.851,-104.321,168.033,47.410,158.821
C00681=1025.629,92.603,-104.303,168.031,47.414,158.822
C00682=1025.624,92.353,-104.284,168.028,47.417,158.822
C00683=1025.617,92.118,-104.267,168.026,47.421,158.822
C00684=1025.612,91.882,-104.249,168.023,47.425,158.823
C00685=1025.607,91.646,-104.232,168.021,47.428,158.823
C00686=1025.601,91.411,-104.214,168.018,47.431,158.823
C00687=1025.595,91.175,-104.197,168.016,47.435,158.824
C00688=1025.590,90.939,-104.180,168.013,47.439,158.824
C00689=1025.584,90.703,-104.163,168.011,47.442,158.825
C00690=1025.579,90.468,-104.145,168.008,47.445,158.825
C00691=1025.573,90.218,-104.126,168.005,47.449,158.825
C00692=1025.567,89.969,-104.108,168.004,47.453,158.826
C00693=1025.561,89.720,-104.089,168.001,47.456,158.826
C00694=1025.556,89.470,-104.071,167.998,47.460,158.826
C00695=1025.550,89.222,-104.052,167.996,47.464,158.827
C00696=1025.544,88.972,-104.034,167.993,47.467,158.827
C00697=1025.537,88.723,-104.016,167.990,47.471,158.828
C00698=1025.532,88.474,-103.998,167.987,47.475,158.828
C00699=1025.526,88.224,-103.980,167.986,47.479,158.828
C00700=1025.519,87.975,-103.962,167.983,47.482,158.829
C00701=1025.513,87.725,-103.944,167.980,47.486,158.829
C00702=1025.507,87.477,-103.925,167.977,47.490,158.829
C00703=1025.501,87.227,-103.907,167.975,47.493,158.830
C00704=1025.495,86.978,-103.889,167.972,47.497,158.830
C00705=1025.489,86.729,-103.871,167.969,47.501,158.831
C00706=1025.483,86.479,-103.853,167.967,47.505,158.831
C00707=1025.477,86.230,-103.835,167.965,47.509,158.831
C00708=1025.471,85.981,-103.817,167.962,47.513,158.832
C00709=1025.465,85.732,-103.798,167.959,47.517,158.832
C00710=1025.460,85.483,-103.780,167.957,47.520,158.833
C00711=1025.454,85.233,-103.762,167.955,47.524,158.833
C00712=1025.447,84.984,-103.744,167.952,47.528,158.833
C00713=1025.442,84.735,-103.726,167.949,47.531,158.834
C00714=1025.436,84.485,-103.708,167.947,47.535,158.834
C00715=1025.429,84.236,-103.690,167.944,47.539,158.834
C00716=1025.424,83.987,-103.672,167.941,47.543,158.835
C00717=1025.418,83.737,-103.654,167.939,47.546,158.835
C00718=1025.412,83.489,-103.636,167.936,47.550,158.836
C00719=1025.406,83.239,-103.618,167.934,47.554,158.836
C00720=1025.400,82.989,-103.600,167.931,47.557,158.836
C00721=1025.394,82.741,-103.582,167.929,47.561,158.837
C00722=1025.388,82.491,-103.564,167.926,47.565,158.837
C00723=1025.382,82.242,-103.546,167.923,47.569,158.837
C00724=1025.376,81.993,-103.527,167.921,47.572,158.838
C00725=1025.370,81.744,-103.510,167.919,47.576,158.838
C00726=1025.364,81.494,-103.492,167.916,47.580,158.839
C00727=1025.357,81.183,-103.469,167.913,47.584,158.839
C00728=1025.349,80.871,-103.446,167.910,47.589,158.840
C00729=1025.342,80.560,-103.424,167.906,47.594,158.840
C00730=1025.334,80.247,-103.402,167.903,47.598,158.841
C00731=1025.329,79.999,-103.384,167.901,47.602,158.841
C00732=1025.323,79.749,-103.365,167.898,47.606,158.841
C00733=1025.318,79.500,-103.348,167.896,47.609,158.842
C00734=1025.312,79.250,-103.330,167.893,47.612,158.842
C00735=1025.306,79.001,-103.312,167.890,47.616,158.842
C00736=1025.300,78.752,-103.294,167.888,47.620,158.843
C00737=1025.293,78.502,-103.276,167.885,47.624,158.843
C00738=1025.288,78.253,-103.258,167.882,47.627,158.843
C00739=1025.282,78.003,-103.240,167.880,47.631,158.844
C00740=1025.276,77.754,-103.223,167.878,47.635,158.844
C00741=1025.270,77.505,-103.205,167.875,47.638,158.845
C00742=1025.264,77.256,-103.187,167.873,47.642,158.845
C00743=1025.257,77.007,-103.169,167.870,47.646,158.845
C00744=1025.252,76.758,-103.152,167.867,47.650,158.846
C00745=1025.246,76.508,-103.134,167.865,47.653,158.846
C00746=1025.240,76.259,-103.116,167.862,47.657,158.846
C00747=1025.234,75.974,-103.096,167.860,47.661,158.847
C00748=1025.226,75.690,-103.076,167.856,47.666,158.847
C00749=1025.220,75.406,-103.056,167.853,47.670,158.848
C00750=1025.213,75.121,-103.036,167.851,47.675,158.848
C00751=1025.207,74.872,-103.018,167.848,47.678,158.849
C00752=1025.201,74.622,-103.001,167.845,47.682,158.849
C00753=1025.195,74.373,-102.983,167.843,47.686,158.849
C00754=1025.189,74.124,-102.965,167.841,47.689,158.850
C00755=1025.183,73.875,-102.948,167.838,47.693,158.850
C00756=1025.177,73.625,-102.930,167.836,47.697,158.851
C00757=1025.171,73.376,-102.913,167.833,47.701,158.851
C00758=1025.165,73.126,-102.895,167.830,47.704,158.851
C00759=1025.159,72.877,-102.877,167.827,47.708,158.852
C00760=1025.152,72.628,-102.860,167.825,47.712,158.852
C00761=1025.147,72.379,-102.842,167.823,47.716,158.852
C00762=1025.142,72.129,-102.825,167.820,47.719,158.853
C00763=1025.136,71.880,-102.807,167.818,47.723,158.853
C00764=1025.129,71.631,-102.791,167.815,47.727,158.853
C00765=1025.123,71.381,-102.773,167.812,47.731,158.854
C00766=1025.118,71.132,-102.755,167.810,47.734,158.854
C00767=1025.111,70.883,-102.738,167.808,47.738,158.855
C00768=1025.105,70.634,-102.720,167.805,47.742,158.855
C00769=1025.100,70.384,-102.703,167.802,47.746,158.855
C00770=1025.094,70.135,-102.685,167.800,47.749,158.856
C00771=1025.088,69.885,-102.668,167.797,47.753,158.856
C00772=1025.082,69.636,-102.650,167.794,47.757,158.856
C00773=1025.076,69.387,-102.633,167.792,47.760,158.857
C00774=1025.069,69.137,-102.616,167.790,47.764,158.857
C00775=1025.064,68.888,-102.598,167.787,47.768,158.858
C00776=1025.058,68.639,-102.580,167.785,47.771,158.858
C00777=1025.052,68.389,-102.564,167.782,47.775,158.858
C00778=1025.046,68.140,-102.546,167.779,47.779,158.859
C00779=1025.039,67.891,-102.529,167.776,47.783,158.859
C00780=1025.034,67.642,-102.511,167.775,47.787,158.859
C00781=1025.029,67.392,-102.494,167.772,47.790,158.860
C00782=1025.022,67.142,-102.477,167.769,47.794,158.860
C00783=1025.016,66.893,-102.460,167.767,47.798,158.861
C00784=1025.010,66.645,-102.443,167.764,47.802,158.861
C00785=1025.004,66.394,-102.425,167.761,47.805,158.861
C00786=1024.998,66.146,-102.408,167.759,47.809,158.862
C00787=1024.992,65.897,-102.391,167.757,47.813,158.862
C00788=1024.986,65.647,-102.374,167.754,47.817,158.862
C00789=1024.980,65.397,-102.357,167.751,47.820,158.863
C00790=1024.973,65.148,-102.339,167.749,47.824,158.863
C00791=1024.968,64.898,-102.322,167.746,47.828,158.864
C00792=1024.962,64.650,-102.305,167.743,47.832,158.864
C00793=1024.956,64.400,-102.288,167.741,47.835,158.864
C00794=1024.950,64.151,-102.271,167.739,47.839,158.865
C00795=1024.944,63.902,-102.254,167.736,47.843,158.865
C00796=1024.938,63.652,-102.236,167.733,47.847,158.865
C00797=1024.932,63.402,-102.219,167.731,47.850,158.866
C00798=1024.926,63.154,-102.203,167.728,47.854,158.866
C00799=1024.920,62.903,-102.185,167.726,47.859,158.867
C00800=1024.914,62.655,-102.168,167.723,47.862,158.867
C00801=1024.908,62.405,-102.152,167.720,47.866,158.867
C00802=1024.901,62.156,-102.135,167.718,47.870,158.868
C00803=1024.895,61.906,-102.118,167.716,47.874,158.868
C00804=1024.890,61.657,-102.101,167.713,47.878,158.869
C00805=1024.883,61.407,-102.084,167.710,47.882,158.869
C00806=1024.877,61.159,-102.067,167.708,47.885,158.869
C00807=1024.871,60.909,-102.051,167.706,47.889,158.870
C00808=1024.865,60.659,-102.034,167.703,47.893,158.870
C00809=1024.859,60.410,-102.017,167.700,47.897,158.870
C00810=1024.853,60.161,-102.001,167.697,47.901,158.871
C00811=1024.846,59.877,-101.981,167.695,47.905,158.871
C00812=1024.838,59.592,-101.962,167.692,47.910,158.872
C00813=1024.831,59.307,-101.943,167.689,47.914,158.872
C00814=1024.825,59.023,-101.924,167.686,47.918,158.873
C00815=1024.819,58.773,-101.906,167.684,47.922,158.873
C00816=1024.813,58.524,-101.890,167.681,47.927,158.874
C00817=1024.807,58.274,-101.874,167.678,47.930,158.874
C00818=1024.800,58.025,-101.857,167.676,47.934,158.874
C00819=1024.794,57.775,-101.840,167.673,47.938,158.875
C00820=1024.788,57.526,-101.823,167.671,47.942,158.875
C00821=1024.782,57.277,-101.806,167.668,47.945,158.875
C00822=1024.776,57.027,-101.790,167.665,47.949,158.876
C00823=1024.770,56.778,-101.773,167.662,47.953,158.876
C00824=1024.764,56.529,-101.757,167.661,47.957,158.877
C00825=1024.759,56.279,-101.740,167.658,47.961,158.877
C00826=1024.752,56.030,-101.722,167.655,47.964,158.877
C00827=1024.746,55.780,-101.706,167.652,47.969,158.878
C00828=1024.740,55.531,-101.690,167.651,47.973,158.878
C00829=1024.733,55.282,-101.673,167.648,47.976,158.878
C00830=1024.728,55.033,-101.657,167.645,47.980,158.879
C00831=1024.722,54.783,-101.639,167.643,47.984,158.879
C00832=1024.716,54.533,-101.623,167.640,47.988,158.880
C00833=1024.710,54.285,-101.606,167.637,47.991,158.880
C00834=1024.704,54.035,-101.590,167.635,47.995,158.880
C00835=1024.698,53.786,-101.574,167.633,47.999,158.881
C00836=1024.692,53.536,-101.556,167.630,48.003,158.881
C00837=1024.686,53.287,-101.540,167.627,48.007,158.881
C00838=1024.680,53.037,-101.523,167.624,48.010,158.882
C00839=1024.674,52.788,-101.507,167.623,48.014,158.882
C00840=1024.668,52.539,-101.491,167.620,48.018,158.883
C00841=1024.661,52.290,-101.474,167.617,48.022,158.883
C00842=1024.656,52.040,-101.457,167.614,48.026,158.883
C00843=1024.650,51.790,-101.440,167.612,48.029,158.884
C00844=1024.644,51.541,-101.424,167.609,48.033,158.884
C00845=1024.637,51.292,-101.407,167.607,48.037,158.884
C00846=1024.632,51.043,-101.391,167.605,48.040,158.885
C00847=1024.626,50.794,-101.375,167.602,48.044,158.885
C00848=1024.620,50.544,-101.358,167.599,48.048,158.885
C00849=1024.614,50.294,-101.341,167.596,48.052,158.886
C00850=1024.608,50.044,-101.325,167.594,48.056,158.886
C00851=1024.602,49.796,-101.308,167.592,48.059,158.887
C00852=1024.596,49.546,-101.292,167.589,48.063,158.887
C00853=1024.590,49.297,-101.275,167.587,48.067,158.887
C00854=1024.584,49.047,-101.258,167.584,48.071,158.888
C00855=1024.579,48.798,-101.242,167.581,48.074,158.888
C00856=1024.573,48.549,-101.226,167.580,48.078,158.888
C00857=1024.566,48.300,-101.209,167.577,48.082,158.889
C00858=1024.560,48.051,-101.193,167.574,48.086,158.889
C00859=1024.554,47.801,-101.176,167.571,48.089,158.889
C00860=1024.549,47.551,-101.159,167.569,48.093,158.890
C00861=1024.543,47.302,-101.143,167.566,48.096,158.890
C00862=1024.537,47.052,-101.127,167.563,48.100,158.890
C00863=1024.531,46.803,-101.111,167.561,48.104,158.891
C00864=1024.525,46.553,-101.094,167.559,48.108,158.891
C00865=1024.519,46.304,-101.078,167.556,48.112,158.891
C00866=1024.514,46.054,-101.061,167.554,48.115,158.892
C00867=1024.508,45.805,-101.045,167.551,48.119,158.892
C00868=1024.502,45.556,-101.029,167.548,48.123,158.893
C00869=1024.495,45.307,-101.012,167.546,48.126,158.893
C00870=1024.490,45.058,-100.995,167.543,48.130,158.893
C00871=1024.484,44.808,-100.979,167.541,48.133,158.893
C00872=1024.478,44.559,-100.963,167.538,48.137,158.894
C00873=1024.472,44.309,-100.946,167.536,48.141,158.894
C00874=1024.466,44.060,-100.930,167.533,48.145,158.895
C00875=1024.460,43.774,-100.912,167.530,48.149,158.895
C00876=1024.453,43.490,-100.893,167.528,48.153,158.895
C00877=1024.446,43.205,-100.874,167.525,48.157,158.896
C00878=1024.439,42.920,-100.856,167.521,48.161,158.896
C00879=1024.433,42.671,-100.839,167.519,48.165,158.896
C00880=1024.427,42.421,-100.823,167.517,48.169,158.897
C00881=1024.421,42.172,-100.807,167.514,48.173,158.897
C00882=1024.415,41.922,-100.791,167.511,48.176,158.897
C00883=1024.410,41.673,-100.774,167.509,48.180,158.898
C00884=1024.404,41.423,-100.759,167.506,48.184,158.898
C00885=1024.398,41.174,-100.743,167.503,48.188,158.899
C00886=1024.391,40.925,-100.727,167.501,48.192,158.899
C00887=1024.385,40.675,-100.711,167.499,48.195,158.899
C00888=1024.379,40.426,-100.694,167.496,48.199,158.900
C00889=1024.373,40.177,-100.678,167.493,48.203,158.900
C00890=1024.368,39.927,-100.663,167.490,48.207,158.900
C00891=1024.362,39.677,-100.646,167.489,48.210,158.901
C00892=1024.356,39.428,-100.630,167.486,48.214,158.901
C00893=1024.350,39.179,-100.614,167.483,48.218,158.901
C00894=1024.343,38.930,-100.598,167.480,48.222,158.902
C00895=1024.338,38.680,-100.583,167.478,48.226,158.902
C00896=1024.332,38.430,-100.566,167.475,48.229,158.903
C00897=1024.326,38.181,-100.550,167.473,48.233,158.903
C00898=1024.320,37.932,-100.534,167.471,48.237,158.903
C00899=1024.315,37.682,-100.519,167.468,48.241,158.904
C00900=1024.309,37.433,-100.502,167.465,48.245,158.904
C00901=1024.302,37.184,-100.487,167.462,48.249,158.904
C00902=1024.296,36.935,-100.470,167.461,48.252,158.905
C00903=1024.290,36.685,-100.455,167.458,48.256,158.905
C00904=1024.284,36.435,-100.439,167.455,48.260,158.905
C00905=1024.278,36.186,-100.424,167.452,48.264,158.906
C00906=1024.272,35.936,-100.407,167.449,48.268,158.906
C00907=1024.265,35.687,-100.392,167.448,48.271,158.906
C00908=1024.260,35.437,-100.376,167.445,48.275,158.907
C00909=1024.254,35.188,-100.360,167.442,48.279,158.907
C00910=1024.247,34.938,-100.345,167.439,48.283,158.907
C00911=1024.241,34.689,-100.329,167.437,48.286,158.908
C00912=1024.236,34.440,-100.313,167.435,48.290,158.908
C00913=1024.230,34.191,-100.298,167.432,48.294,158.909
C00914=1024.224,33.941,-100.282,167.429,48.298,158.909
C00915=1024.217,33.692,-100.267,167.426,48.302,158.909
C00916=1024.211,33.442,-100.251,167.424,48.306,158.910
C00917=1024.206,33.192,-100.235,167.421,48.309,158.910
C00918=1024.199,32.943,-100.219,167.419,48.313,158.910
C00919=1024.193,32.693,-100.204,167.416,48.317,158.911
C00920=1024.187,32.444,-100.188,167.414,48.321,158.911
C00921=1024.181,32.195,-100.172,167.411,48.325,158.911
C00922=1024.176,31.946,-100.157,167.408,48.329,158.912
C00923=1024.169,31.697,-100.141,167.406,48.332,158.912
C00924=1024.163,31.447,-100.125,167.403,48.336,158.912
C00925=1024.157,31.198,-100.110,167.401,48.340,158.913
C00926=1024.151,30.948,-100.094,167.398,48.344,158.913
C00927=1024.146,30.698,-100.079,167.395,48.348,158.914
C00928=1024.139,30.449,-100.063,167.393,48.352,158.914
C00929=1024.134,30.199,-100.048,167.391,48.355,158.914
C00930=1024.128,29.950,-100.032,167.388,48.359,158.915
C00931=1024.121,29.700,-100.017,167.385,48.363,158.915
C00932=1024.115,29.451,-100.000,167.382,48.367,158.915
C00933=1024.109,29.201,-99.985,167.381,48.370,158.916
C00934=1024.104,28.953,-99.970,167.377,48.374,158.916
C00935=1024.097,28.703,-99.955,167.375,48.378,158.916
C00936=1024.092,28.453,-99.939,167.372,48.381,158.917
C00937=1024.086,28.204,-99.923,167.369,48.385,158.917
C00938=1024.079,27.954,-99.908,167.367,48.389,158.917
C00939=1024.073,27.669,-99.890,167.364,48.394,158.918
C00940=1024.066,27.385,-99.873,167.361,48.398,158.918
C00941=1024.059,27.100,-99.855,167.358,48.402,158.919
C00942=1024.053,26.815,-99.837,167.355,48.406,158.919
C00943=1024.046,26.565,-99.822,167.353,48.410,158.919
C00944=1024.039,26.316,-99.807,167.350,48.414,158.919
C00945=1024.034,26.067,-99.791,167.347,48.418,158.920
C00946=1024.028,25.817,-99.776,167.344,48.422,158.920
C00947=1024.022,25.567,-99.761,167.342,48.426,158.920
C00948=1024.016,25.318,-99.745,167.339,48.430,158.921
C00949=1024.010,25.069,-99.731,167.337,48.433,158.921
C00950=1024.004,24.819,-99.715,167.334,48.437,158.922
C00951=1023.998,24.570,-99.700,167.332,48.442,158.922
C00952=1023.991,24.320,-99.685,167.329,48.446,158.922
C00953=1023.986,24.071,-99.669,167.326,48.449,158.923
C00954=1023.980,23.822,-99.654,167.324,48.453,158.923
C00955=1023.973,23.572,-99.639,167.321,48.456,158.923
C00956=1023.968,23.322,-99.624,167.318,48.460,158.924
C00957=1023.962,23.073,-99.609,167.316,48.464,158.924
C00958=1023.956,22.824,-99.593,167.313,48.468,158.924
C00959=1023.950,22.574,-99.578,167.311,48.472,158.925
C00960=1023.943,22.324,-99.563,167.308,48.475,158.925
C00961=1023.938,22.075,-99.548,167.305,48.479,158.925
C00962=1023.932,21.825,-99.533,167.303,48.483,158.926
C00963=1023.925,21.576,-99.518,167.300,48.487,158.926
C00964=1023.920,21.327,-99.502,167.298,48.491,158.926
C00965=1023.914,21.077,-99.487,167.295,48.495,158.927
C00966=1023.907,20.828,-99.472,167.292,48.499,158.927
C00967=1023.902,20.578,-99.457,167.290,48.503,158.927
C00968=1023.896,20.329,-99.442,167.287,48.506,158.928
C00969=1023.889,20.079,-99.427,167.285,48.510,158.928
C00970=1023.884,19.829,-99.412,167.282,48.514,158.929
C00971=1023.878,19.580,-99.397,167.279,48.518,158.929
C00972=1023.872,19.331,-99.382,167.277,48.522,158.929
C00973=1023.866,19.081,-99.367,167.274,48.526,158.929
C00974=1023.860,18.832,-99.352,167.271,48.530,158.930
C00975=1023.854,18.582,-99.337,167.269,48.533,158.930
C00976=1023.847,18.332,-99.322,167.267,48.537,158.931
C00977=1023.842,18.083,-99.308,167.264,48.541,158.931
C00978=1023.836,17.833,-99.292,167.261,48.545,158.931
C00979=1023.830,17.584,-99.277,167.258,48.549,158.932
C00980=1023.824,17.335,-99.262,167.255,48.552,158.932
C00981=1023.818,17.085,-99.248,167.253,48.556,158.932
C00982=1023.811,16.836,-99.233,167.250,48.560,158.932
C00983=1023.806,16.586,-99.217,167.248,48.563,158.933
C00984=1023.800,16.337,-99.202,167.245,48.567,158.933
C00985=1023.794,16.088,-99.188,167.242,48.571,158.933
C00986=1023.788,15.838,-99.173,167.239,48.575,158.934
C00987=1023.781,15.588,-99.158,167.237,48.579,158.934
C00988=1023.775,15.339,-99.143,167.235,48.583,158.934
C00989=1023.770,15.089,-99.128,167.232,48.587,158.935
C00990=1023.764,14.840,-99.113,167.229,48.591,158.935
C00991=1023.758,14.591,-99.098,167.226,48.595,158.935
C00992=1023.751,14.341,-99.083,167.225,48.598,158.936
C00993=1023.745,14.092,-99.069,167.222,48.602,158.936
C00994=1023.740,13.842,-99.054,167.219,48.606,158.937
C00995=1023.734,13.593,-99.039,167.216,48.609,158.937
C00996=1023.728,13.343,-99.024,167.213,48.614,158.937
C00997=1023.722,13.093,-99.010,167.211,48.618,158.938
C00998=1023.716,12.844,-98.995,167.208,48.622,158.938
C00999=1023.710,12.594,-98.981,167.205,48.626,158.938
C01000=1023.703,12.345,-98.967,167.203,48.629,158.939
C01001=1023.697,12.096,-98.952,167.200,48.633,158.939
C01002=1023.691,11.846,-98.938,167.198,48.637,158.939
C01003=1023.683,11.563,-98.920,167.194,48.642,158.940
C01004=1023.678,11.280,-98.904,167.191,48.646,158.940
C01005=1023.670,10.996,-98.888,167.188,48.651,158.940
C01006=1023.663,10.713,-98.871,167.185,48.655,158.941
C01007=1023.657,10.462,-98.857,167.182,48.659,158.941
C01008=1023.652,10.213,-98.842,167.179,48.662,158.941
C01009=1023.645,9.964,-98.827,167.177,48.666,158.942
C01010=1023.639,9.713,-98.813,167.174,48.670,158.942
C01011=1023.633,9.465,-98.799,167.172,48.674,158.942
C01012=1023.626,9.215,-98.784,167.169,48.678,158.943
C01013=1023.621,8.966,-98.770,167.167,48.682,158.943
C01014=1023.614,8.716,-98.755,167.164,48.686,158.943
C01015=1023.609,8.467,-98.741,167.161,48.690,158.944
C01016=1023.602,8.217,-98.727,167.158,48.694,158.944
C01017=1023.597,7.968,-98.712,167.155,48.698,158.944
C01018=1023.590,7.718,-98.697,167.153,48.701,158.945
C01019=1023.585,7.469,-98.683,167.150,48.705,158.945
C01020=1023.578,7.219,-98.668,167.148,48.709,158.945
C01021=1023.573,6.969,-98.654,167.145,48.713,158.946
C01022=1023.566,6.720,-98.640,167.142,48.717,158.946
C01023=1023.560,6.470,-98.626,167.140,48.721,158.946
C01024=1023.554,6.221,-98.611,167.137,48.725,158.947
C01025=1023.548,5.972,-98.597,167.134,48.729,158.947
C01026=1023.543,5.722,-98.583,167.131,48.733,158.947
C01027=1023.536,5.473,-98.568,167.129,48.737,158.948
C01028=1023.531,5.223,-98.554,167.126,48.740,158.948
C01029=1023.524,4.973,-98.539,167.124,48.744,158.948
C01030=1023.518,4.724,-98.526,167.121,48.748,158.949
C01031=1023.512,4.474,-98.511,167.118,48.752,158.949
C01032=1023.506,4.225,-98.497,167.116,48.756,158.949
C01033=1023.500,3.975,-98.482,167.113,48.760,158.950
C01034=1023.495,3.726,-98.468,167.110,48.763,158.950
C01035=1023.489,3.477,-98.454,167.107,48.767,158.950
C01036=1023.483,3.226,-98.439,167.104,48.771,158.950
C01037=1023.477,2.977,-98.425,167.102,48.775,158.951
C01038=1023.471,2.727,-98.411,167.100,48.779,158.951
C01039=1023.464,2.478,-98.397,167.097,48.782,158.951
C01040=1023.459,2.229,-98.383,167.094,48.786,158.952
C01041=1023.452,1.979,-98.368,167.091,48.790,158.952
C01042=1023.447,1.730,-98.354,167.089,48.794,158.952
C01043=1023.441,1.481,-98.339,167.085,48.797,158.953
C01044=1023.435,1.230,-98.325,167.083,48.801,158.953
C01045=1023.430,0.981,-98.311,167.081,48.805,158.953
C01046=1023.423,0.732,-98.297,167.078,48.809,158.954
C01047=1023.417,0.482,-98.283,167.075,48.813,158.954
C01048=1023.411,0.233,-98.268,167.073,48.817,158.954
C01049=1023.405,-0.017,-98.254,167.069,48.820,158.954
C01050=1023.400,-0.267,-98.240,167.067,48.824,158.955
C01051=1023.394,-0.516,-98.226,167.064,48.828,158.955
C01052=1023.388,-0.766,-98.212,167.062,48.832,158.955
C01053=1023.382,-1.015,-98.197,167.059,48.836,158.956
C01054=1023.376,-1.264,-98.184,167.057,48.840,158.956
C01055=1023.370,-1.515,-98.169,167.053,48.843,158.956
C01056=1023.364,-1.764,-98.155,167.051,48.847,158.957
C01057=1023.359,-2.013,-98.141,167.048,48.851,158.957
C01058=1023.352,-2.263,-98.127,167.045,48.855,158.957
C01059=1023.347,-2.512,-98.112,167.043,48.858,158.958
C01060=1023.340,-2.762,-98.099,167.040,48.862,158.958
C01061=1023.335,-3.011,-98.085,167.037,48.865,158.958
C01062=1023.329,-3.261,-98.070,167.035,48.869,158.958
C01063=1023.323,-3.510,-98.056,167.032,48.873,158.959
C01064=1023.318,-3.760,-98.042,167.029,48.877,158.959
C01065=1023.312,-4.010,-98.028,167.026,48.881,158.959
C01066=1023.305,-4.260,-98.015,167.023,48.884,158.959
C01067=1023.299,-4.541,-97.999,167.021,48.889,158.960
C01068=1023.292,-4.822,-97.983,167.018,48.893,158.960
C01069=1023.285,-5.105,-97.967,167.015,48.898,158.961
C01070=1023.278,-5.386,-97.952,167.012,48.902,158.961
C01071=1023.272,-5.635,-97.938,167.009,48.906,158.961
C01072=1023.266,-5.884,-97.925,167.006,48.910,158.962
C01073=1023.260,-6.134,-97.911,167.003,48.914,158.962
C01074=1023.254,-6.384,-97.897,167.001,48.918,158.962
C01075=1023.248,-6.633,-97.884,166.998,48.922,158.963
C01076=1023.242,-6.883,-97.870,166.995,48.926,158.963
C01077=1023.236,-7.133,-97.856,166.992,48.930,158.963
C01078=1023.230,-7.382,-97.842,166.990,48.934,158.964
C01079=1023.224,-7.632,-97.829,166.987,48.938,158.964
C01080=1023.218,-7.881,-97.815,166.984,48.941,158.964
C01081=1023.212,-8.131,-97.802,166.981,48.945,158.964
C01082=1023.206,-8.381,-97.788,166.978,48.949,158.965
C01083=1023.200,-8.630,-97.775,166.975,48.953,158.965
C01084=1023.194,-8.880,-97.761,166.973,48.957,158.965
C01085=1023.188,-9.129,-97.747,166.970,48.961,158.966
C01086=1023.182,-9.379,-97.733,166.967,48.965,158.966
C01087=1023.176,-9.628,-97.720,166.964,48.968,158.966
C01088=1023.170,-9.878,-97.706,166.961,48.972,158.966
C01089=1023.164,-10.127,-97.693,166.959,48.976,158.967
C01090=1023.159,-10.377,-97.679,166.956,48.980,158.967
C01091=1023.152,-10.627,-97.665,166.953,48.984,158.967
C01092=1023.146,-10.876,-97.651,166.951,48.988,158.968
C01093=1023.140,-11.126,-97.638,166.948,48.991,158.968
C01094=1023.135,-11.375,-97.624,166.946,48.995,158.968
C01095=1023.129,-11.624,-97.611,166.943,48.999,158.969
C01096=1023.123,-11.874,-97.597,166.940,49.003,158.969
C01097=1023.116,-12.124,-97.583,166.937,49.007,158.969
C01098=1023.111,-12.374,-97.570,166.934,49.011,158.970
C01099=1023.105,-12.623,-97.556,166.932,49.015,158.970
C01100=1023.098,-12.872,-97.543,166.929,49.018,158.970
C01101=1023.093,-13.122,-97.530,166.926,49.022,158.970
C01102=1023.087,-13.372,-97.517,166.923,49.026,158.971
C01103=1023.082,-13.621,-97.503,166.920,49.030,158.971
C01104=1023.075,-13.870,-97.490,166.918,49.034,158.971
C01105=1023.069,-14.121,-97.475,166.915,49.038,158.972
C01106=1023.063,-14.370,-97.462,166.912,49.041,158.972
C01107=1023.058,-14.620,-97.448,166.909,49.045,158.972
C01108=1023.051,-14.869,-97.435,166.906,49.049,158.972
C01109=1023.046,-15.119,-97.422,166.904,49.053,158.973
C01110=1023.040,-15.368,-97.408,166.902,49.057,158.973
C01111=1023.034,-15.618,-97.395,166.899,49.060,158.973
C01112=1023.028,-15.867,-97.381,166.896,49.064,158.973
C01113=1023.022,-16.117,-97.369,166.893,49.068,158.974
C01114=1023.016,-16.366,-97.356,166.890,49.072,158.974
C01115=1023.010,-16.617,-97.341,166.887,49.076,158.974
C01116=1023.004,-16.866,-97.329,166.885,49.080,158.975
C01117=1022.998,-17.116,-97.315,166.882,49.084,158.975
C01118=1022.992,-17.365,-97.302,166.879,49.088,158.975
C01119=1022.986,-17.615,-97.290,166.876,49.092,158.976
C01120=1022.980,-17.864,-97.276,166.874,49.096,158.976
C01121=1022.974,-18.114,-97.263,166.871,49.100,158.976
C01122=1022.968,-18.364,-97.250,166.868,49.104,158.977
C01123=1022.962,-18.613,-97.237,166.864,49.108,158.977
C01124=1022.956,-18.862,-97.223,166.862,49.112,158.977
C01125=1022.951,-19.112,-97.210,166.858,49.115,158.977
C01126=1022.944,-19.362,-97.197,166.856,49.119,158.977
C01127=1022.938,-19.611,-97.184,166.853,49.123,158.978
C01128=1022.932,-19.861,-97.171,166.850,49.127,158.978
C01129=1022.926,-20.110,-97.158,166.847,49.131,158.978
C01130=1022.921,-20.360,-97.145,166.845,49.135,158.979
C01131=1022.914,-20.640,-97.130,166.842,49.139,158.979
C01132=1022.907,-20.920,-97.116,166.838,49.144,158.979
C01133=1022.900,-21.200,-97.101,166.836,49.148,158.980
C01134=1022.893,-21.480,-97.086,166.832,49.152,158.980
C01135=1022.887,-21.730,-97.073,166.829,49.156,158.980
C01136=1022.882,-21.979,-97.060,166.826,49.160,158.981
C01137=1022.876,-22.229,-97.047,166.824,49.164,158.981
C01138=1022.870,-22.478,-97.034,166.821,49.168,158.981
C01139=1022.864,-22.728,-97.022,166.818,49.172,158.981
C01140=1022.858,-22.977,-97.008,166.815,49.176,158.982
C01141=1022.853,-23.227,-96.995,166.812,49.180,158.982
C01142=1022.847,-23.476,-96.982,166.809,49.184,158.982
C01143=1022.841,-23.726,-96.969,166.807,49.187,158.982
C01144=1022.835,-23.975,-96.956,166.804,49.191,158.983
C01145=1022.829,-24.225,-96.944,166.801,49.195,158.983
C01146=1022.823,-24.475,-96.930,166.798,49.199,158.983
C01147=1022.817,-24.725,-96.917,166.795,49.203,158.984
C01148=1022.811,-24.974,-96.904,166.793,49.207,158.984
C01149=1022.805,-25.224,-96.891,166.790,49.211,158.984
C01150=1022.799,-25.473,-96.878,166.787,49.215,158.984
C01151=1022.793,-25.723,-96.865,166.784,49.218,158.985
C01152=1022.788,-25.972,-96.853,166.781,49.222,158.985
C01153=1022.782,-26.222,-96.839,166.778,49.226,158.985
C01154=1022.776,-26.472,-96.827,166.776,49.230,158.985
C01155=1022.770,-26.721,-96.814,166.773,49.233,158.986
C01156=1022.764,-26.971,-96.801,166.770,49.237,158.986
C01157=1022.758,-27.221,-96.788,166.767,49.241,158.986
C01158=1022.752,-27.470,-96.775,166.764,49.245,158.987
C01159=1022.746,-27.720,-96.763,166.762,49.249,158.987
C01160=1022.741,-27.969,-96.750,166.759,49.253,158.987
C01161=1022.735,-28.219,-96.738,166.756,49.257,158.987
C01162=1022.729,-28.468,-96.725,166.753,49.261,158.988
C01163=1022.723,-28.718,-96.712,166.750,49.264,158.988
C01164=1022.717,-28.968,-96.700,166.747,49.268,158.988
C01165=1022.711,-29.218,-96.687,166.745,49.272,158.988
C01166=1022.705,-29.467,-96.674,166.742,49.276,158.989
C01167=1022.699,-29.716,-96.662,166.739,49.280,158.989
C01168=1022.693,-29.966,-96.650,166.736,49.284,158.989
C01169=1022.687,-30.216,-96.637,166.734,49.288,158.990
C01170=1022.681,-30.466,-96.624,166.731,49.292,158.990
C01171=1022.675,-30.715,-96.611,166.727,49.297,158.990
C01172=1022.669,-30.965,-96.599,166.724,49.301,158.990
C01173=1022.664,-31.214,-96.586,166.721,49.304,158.991
C01174=1022.658,-31.464,-96.574,166.719,49.308,158.991
C01175=1022.652,-31.714,-96.561,166.716,49.312,158.991
C01176=1022.645,-31.963,-96.549,166.713,49.316,158.992
C01177=1022.639,-32.213,-96.537,166.710,49.320,158.992
C01178=1022.634,-32.462,-96.524,166.708,49.324,158.992
C01179=1022.628,-32.712,-96.511,166.705,49.328,158.992
C01180=1022.622,-32.961,-96.499,166.702,49.332,158.993
C01181=1022.616,-33.211,-96.486,166.699,49.335,158.993
C01182=1022.611,-33.461,-96.474,166.696,49.339,158.993
C01183=1022.605,-33.710,-96.462,166.693,49.343,158.993
C01184=1022.598,-33.960,-96.450,166.691,49.347,158.994
C01185=1022.592,-34.210,-96.437,166.688,49.351,158.994
C01186=1022.587,-34.459,-96.425,166.684,49.355,158.994
C01187=1022.581,-34.709,-96.412,166.681,49.359,158.994
C01188=1022.575,-34.959,-96.400,166.678,49.363,158.995
C01189=1022.569,-35.209,-96.387,166.676,49.367,158.995
C01190=1022.564,-35.458,-96.375,166.673,49.371,158.995
C01191=1022.557,-35.707,-96.363,166.670,49.375,158.996
C01192=1022.551,-35.957,-96.350,166.667,49.378,158.996
C01193=1022.546,-36.207,-96.338,166.664,49.382,158.996
C01194=1022.540,-36.456,-96.326,166.661,49.386,158.996
C01195=1022.534,-36.736,-96.311,166.658,49.390,158.996
C01196=1022.527,-37.014,-96.298,166.655,49.394,158.997
C01197=1022.521,-37.294,-96.283,166.652,49.399,158.997
C01198=1022.514,-37.572,-96.270,166.649,49.403,158.997
C01199=1022.508,-37.822,-96.257,166.646,49.407,158.998
C01200=1022.502,-38.072,-96.246,166.643,49.411,158.998
C01201=1022.497,-38.321,-96.233,166.640,49.415,158.998
C01202=1022.491,-38.571,-96.221,166.637,49.419,158.998
C01203=1022.485,-38.821,-96.209,166.635,49.423,158.999
C01204=1022.479,-39.070,-96.197,166.632,49.426,158.999
C01205=1022.473,-39.320,-96.184,166.628,49.430,158.999
C01206=1022.468,-39.570,-96.172,166.625,49.434,158.999
C01207=1022.461,-39.819,-96.160,166.622,49.438,159.000
C01208=1022.456,-40.069,-96.148,166.620,49.442,159.000
C01209=1022.449,-40.319,-96.136,166.617,49.446,159.000
C01210=1022.444,-40.568,-96.124,166.614,49.450,159.001
C01211=1022.437,-40.818,-96.112,166.611,49.454,159.001
C01212=1022.432,-41.067,-96.101,166.609,49.458,159.001
C01213=1022.426,-41.317,-96.088,166.605,49.462,159.001
C01214=1022.420,-41.567,-96.076,166.602,49.466,159.001
C01215=1022.414,-41.816,-96.064,166.599,49.470,159.002
C01216=1022.408,-42.066,-96.053,166.596,49.474,159.002
C01217=1022.403,-42.315,-96.040,166.594,49.478,159.002
C01218=1022.397,-42.565,-96.028,166.591,49.482,159.003
C01219=1022.390,-42.815,-96.016,166.588,49.486,159.003
C01220=1022.385,-43.065,-96.004,166.584,49.490,159.003
C01221=1022.379,-43.314,-95.993,166.581,49.494,159.003
C01222=1022.373,-43.563,-95.980,166.578,49.498,159.004
C01223=1022.368,-43.814,-95.968,166.576,49.502,159.004
C01224=1022.362,-44.063,-95.957,166.573,49.506,159.004
C01225=1022.356,-44.313,-95.944,166.570,49.510,159.004
C01226=1022.349,-44.563,-95.933,166.568,49.514,159.005
C01227=1022.344,-44.812,-95.921,166.564,49.517,159.005
C01228=1022.337,-45.062,-95.909,166.562,49.521,159.005
C01229=1022.332,-45.311,-95.897,166.558,49.525,159.005
C01230=1022.326,-45.561,-95.885,166.555,49.529,159.006
C01231=1022.321,-45.811,-95.874,166.552,49.533,159.006
C01232=1022.315,-46.061,-95.862,166.550,49.537,159.006
C01233=1022.309,-46.309,-95.850,166.547,49.541,159.006
C01234=1022.303,-46.560,-95.838,166.544,49.545,159.007
C01235=1022.297,-46.809,-95.826,166.541,49.549,159.007
C01236=1022.292,-47.059,-95.815,166.538,49.553,159.007
C01237=1022.285,-47.308,-95.803,166.535,49.557,159.007
C01238=1022.280,-47.558,-95.790,166.532,49.560,159.007
C01239=1022.275,-47.808,-95.779,166.529,49.564,159.008
C01240=1022.268,-48.057,-95.767,166.526,49.568,159.008
C01241=1022.263,-48.307,-95.756,166.523,49.573,159.008
C01242=1022.256,-48.557,-95.744,166.520,49.576,159.008
C01243=1022.251,-48.807,-95.732,166.518,49.580,159.009
C01244=1022.245,-49.056,-95.721,166.515,49.584,159.009
C01245=1022.240,-49.306,-95.709,166.512,49.588,159.009
C01246=1022.234,-49.555,-95.697,166.509,49.591,159.009
C01247=1022.228,-49.805,-95.685,166.505,49.596,159.010
C01248=1022.223,-50.055,-95.673,166.502,49.600,159.010
C01249=1022.216,-50.305,-95.662,166.500,49.604,159.010
C01250=1022.211,-50.554,-95.650,166.497,49.607,159.010
C01251=1022.205,-50.804,-95.638,166.494,49.611,159.011
C01252=1022.200,-51.054,-95.627,166.491,49.615,159.011
C01253=1022.194,-51.303,-95.615,166.488,49.619,159.011
C01254=1022.187,-51.553,-95.604,166.485,49.623,159.011
C01255=1022.182,-51.803,-95.593,166.482,49.627,159.012
C01256=1022.175,-52.052,-95.581,166.479,49.631,159.012
C01257=1022.169,-52.302,-95.570,166.476,49.635,159.012
C01258=1022.164,-52.552,-95.559,166.473,49.640,159.012
C01259=1022.157,-52.831,-95.546,166.470,49.644,159.013
C01260=1022.150,-53.110,-95.534,166.467,49.649,159.013
C01261=1022.144,-53.390,-95.521,166.463,49.653,159.013
C01262=1022.137,-53.669,-95.509,166.459,49.658,159.014
C01263=1022.131,-53.919,-95.497,166.457,49.662,159.014
C01264=1022.125,-54.168,-95.486,166.454,49.666,159.014
C01265=1022.119,-54.418,-95.475,166.451,49.670,159.015
C01266=1022.114,-54.668,-95.463,166.448,49.674,159.015
C01267=1022.108,-54.918,-95.452,166.444,49.678,159.015
C01268=1022.102,-55.168,-95.441,166.442,49.682,159.015
C01269=1022.096,-55.417,-95.430,166.439,49.686,159.015
C01270=1022.090,-55.666,-95.418,166.436,49.690,159.016
C01271=1022.083,-55.916,-95.407,166.432,49.694,159.016
C01272=1022.078,-56.166,-95.396,166.430,49.698,159.016
C01273=1022.073,-56.416,-95.385,166.427,49.702,159.016
C01274=1022.066,-56.666,-95.374,166.424,49.707,159.017
C01275=1022.061,-56.915,-95.363,166.421,49.711,159.017
C01276=1022.055,-57.165,-95.352,166.418,49.715,159.017
C01277=1022.049,-57.414,-95.340,166.415,49.719,159.017
C01278=1022.042,-57.664,-95.329,166.412,49.723,159.018
C01279=1022.037,-57.913,-95.318,166.409,49.726,159.018
C01280=1022.032,-58.163,-95.307,166.405,49.731,159.018
C01281=1022.025,-58.413,-95.295,166.403,49.735,159.018
C01282=1022.020,-58.663,-95.285,166.400,49.739,159.019
C01283=1022.014,-58.912,-95.274,166.397,49.743,159.019
C01284=1022.008,-59.162,-95.263,166.395,49.747,159.019
C01285=1022.002,-59.412,-95.252,166.391,49.751,159.019
C01286=1021.996,-59.661,-95.241,166.388,49.755,159.020
C01287=1021.990,-59.911,-95.230,166.385,49.759,159.020
C01288=1021.985,-60.161,-95.218,166.382,49.763,159.020
///RCONF 1,0,0,1,0,0,0,0,0,0,0,0,0,0,0,0,0,0,0,0,0,0,0,0
C01289=1021.979,-60.411,-95.207,166.380,49.767,159.020
C01290=1021.973,-60.660,-95.196,166.376,49.771,159.021
C01291=1021.968,-60.910,-95.185,166.373,49.775,159.021
C01292=1021.962,-61.159,-95.174,166.370,49.779,159.021
C01293=1021.956,-61.409,-95.164,166.368,49.783,159.021
C01294=1021.950,-61.659,-95.152,166.365,49.786,159.021
C01295=1021.944,-61.909,-95.141,166.361,49.791,159.022
C01296=1021.939,-62.158,-95.130,166.358,49.795,159.022
C01297=1021.933,-62.408,-95.119,166.355,49.799,159.022
C01298=1021.928,-62.657,-95.108,166.353,49.803,159.023
C01299=1021.921,-62.908,-95.097,166.350,49.806,159.023
C01300=1021.915,-63.157,-95.086,166.346,49.811,159.023
C01301=1021.910,-63.406,-95.075,166.343,49.815,159.023
C01302=1021.904,-63.656,-95.064,166.340,49.819,159.023
C01303=1021.898,-63.905,-95.053,166.338,49.823,159.024
C01304=1021.894,-64.156,-95.043,166.335,49.826,159.024
C01305=1021.887,-64.406,-95.031,166.331,49.831,159.024
C01306=1021.881,-64.656,-95.021,166.328,49.835,159.024
C01307=1021.876,-64.905,-95.010,166.325,49.839,159.024
C01308=1021.870,-65.155,-94.999,166.322,49.842,159.025
C01309=1021.864,-65.404,-94.988,166.320,49.846,159.025
C01310=1021.858,-65.654,-94.977,166.316,49.850,159.025
C01311=1021.853,-65.904,-94.967,166.313,49.854,159.025
C01312=1021.847,-66.153,-94.956,166.310,49.858,159.026
C01313=1021.842,-66.403,-94.945,166.307,49.862,159.026
C01314=1021.837,-66.652,-94.934,166.305,49.866,159.026
C01315=1021.830,-66.903,-94.922,166.302,49.870,159.026
C01316=1021.824,-67.152,-94.912,166.298,49.874,159.026
C01317=1021.819,-67.402,-94.901,166.295,49.878,159.027
C01318=1021.813,-67.652,-94.891,166.292,49.882,159.027
C01319=1021.808,-67.901,-94.880,166.290,49.886,159.027
C01320=1021.802,-68.151,-94.869,166.286,49.889,159.027
C01321=1021.796,-68.401,-94.859,166.284,49.893,159.027
C01322=1021.791,-68.650,-94.848,166.280,49.898,159.028
C01323=1021.784,-68.931,-94.835,166.277,49.902,159.028
C01324=1021.778,-69.212,-94.824,166.274,49.906,159.028
C01325=1021.772,-69.492,-94.811,166.270,49.910,159.028
C01326=1021.766,-69.773,-94.799,166.267,49.914,159.029
C01327=1021.760,-70.023,-94.788,166.263,49.919,159.029
C01328=1021.754,-70.272,-94.777,166.261,49.923,159.029
C01329=1021.749,-70.522,-94.767,166.258,49.926,159.029
C01330=1021.743,-70.772,-94.756,166.255,49.930,159.029
C01331=1021.738,-71.020,-94.746,166.252,49.934,159.030
C01332=1021.732,-71.271,-94.736,166.249,49.938,159.030
C01333=1021.727,-71.520,-94.725,166.245,49.942,159.030
C01334=1021.721,-71.770,-94.714,166.243,49.946,159.030
C01335=1021.716,-72.020,-94.704,166.239,49.949,159.030
C01336=1021.710,-72.269,-94.693,166.237,49.953,159.031
C01337=1021.704,-72.519,-94.682,166.234,49.958,159.031
C01338=1021.699,-72.769,-94.671,166.231,49.961,159.031
C01339=1021.694,-73.019,-94.660,166.228,49.965,159.031
C01340=1021.688,-73.269,-94.650,166.225,49.969,159.031
C01341=1021.682,-73.518,-94.639,166.221,49.973,159.031
C01342=1021.677,-73.768,-94.628,166.219,49.977,159.032
C01343=1021.671,-74.018,-94.618,166.216,49.980,159.032
C01344=1021.666,-74.267,-94.607,166.213,49.984,159.032
C01345=1021.660,-74.517,-94.597,166.210,49.988,159.032
C01346=1021.654,-74.767,-94.586,166.206,49.993,159.033
C01347=1021.648,-75.017,-94.577,166.203,49.996,159.033
C01348=1021.643,-75.267,-94.567,166.201,50.000,159.033
C01349=1021.637,-75.516,-94.556,166.198,50.004,159.033
C01350=1021.632,-75.766,-94.546,166.194,50.009,159.033
C01351=1021.626,-76.015,-94.535,166.192,50.013,159.034
C01352=1021.620,-76.265,-94.525,166.188,50.016,159.034
C01353=1021.615,-76.515,-94.515,166.186,50.020,159.034
C01354=1021.609,-76.765,-94.504,166.182,50.024,159.034
C01355=1021.604,-77.015,-94.494,166.179,50.028,159.034
C01356=1021.597,-77.264,-94.484,166.177,50.033,159.035
C01357=1021.592,-77.514,-94.474,166.174,50.036,159.035
C01358=1021.587,-77.763,-94.464,166.170,50.040,159.035
C01359=1021.581,-78.013,-94.453,166.167,50.044,159.035
C01360=1021.575,-78.263,-94.444,166.164,50.048,159.036
C01361=1021.570,-78.513,-94.433,166.162,50.053,159.036
C01362=1021.564,-78.762,-94.422,166.159,50.056,159.036
C01363=1021.558,-79.012,-94.412,166.155,50.060,159.036
C01364=1021.553,-79.261,-94.403,166.152,50.064,159.036
C01365=1021.547,-79.512,-94.393,166.149,50.068,159.037
C01366=1021.542,-79.761,-94.382,166.146,50.072,159.037
C01367=1021.536,-80.011,-94.372,166.143,50.076,159.037
C01368=1021.530,-80.261,-94.362,166.140,50.080,159.037
C01369=1021.525,-80.511,-94.352,166.137,50.084,159.037
C01370=1021.519,-80.760,-94.343,166.133,50.089,159.038
C01371=1021.513,-81.010,-94.332,166.131,50.093,159.038
C01372=1021.507,-81.259,-94.323,166.128,50.097,159.038
C01373=1021.502,-81.510,-94.312,166.125,50.100,159.038
C01374=1021.496,-81.759,-94.303,166.121,50.105,159.038
C01375=1021.491,-82.009,-94.293,166.119,50.109,159.039
C01376=1021.485,-82.259,-94.283,166.116,50.113,159.039
C01377=1021.479,-82.509,-94.273,166.112,50.117,159.039
C01378=1021.473,-82.758,-94.264,166.109,50.121,159.039
C01379=1021.468,-83.008,-94.254,166.107,50.125,159.040
C01380=1021.462,-83.257,-94.244,166.103,50.130,159.040
C01381=1021.456,-83.507,-94.234,166.100,50.134,159.040
C01382=1021.450,-83.757,-94.224,166.098,50.138,159.040
C01383=1021.445,-84.006,-94.214,166.093,50.142,159.040
C01384=1021.439,-84.256,-94.205,166.091,50.146,159.041
C01385=1021.434,-84.506,-94.194,166.088,50.150,159.041
C01386=1021.427,-84.756,-94.185,166.085,50.154,159.041
C01387=1021.420,-85.123,-94.171,166.080,50.160,159.041
C01388=1021.411,-85.491,-94.157,166.076,50.166,159.042
C01389=1021.403,-85.839,-94.143,166.072,50.172,159.042
C01390=1021.396,-86.188,-94.129,166.067,50.177,159.042
C01391=1021.388,-86.537,-94.116,166.063,50.183,159.043
C01392=1021.380,-86.885,-94.102,166.059,50.189,159.043
C01393=1021.374,-87.135,-94.092,166.056,50.193,159.043
C01394=1021.368,-87.385,-94.083,166.052,50.197,159.043
C01395=1021.363,-87.634,-94.073,166.049,50.201,159.043
C01396=1021.357,-87.885,-94.064,166.047,50.205,159.044
C01397=1021.352,-88.135,-94.054,166.044,50.209,159.044
C01398=1021.346,-88.384,-94.045,166.040,50.213,159.044
C01399=1021.341,-88.634,-94.034,166.038,50.217,159.044
C01400=1021.335,-88.883,-94.025,166.034,50.221,159.044
C01401=1021.330,-89.133,-94.015,166.031,50.225,159.045
C01402=1021.324,-89.383,-94.005,166.028,50.229,159.045
C01403=1021.318,-89.632,-93.996,166.025,50.233,159.045
C01404=1021.313,-89.883,-93.987,166.023,50.237,159.045
C01405=1021.308,-90.132,-93.978,166.019,50.241,159.045
C01406=1021.302,-90.382,-93.967,166.016,50.245,159.046
C01407=1021.296,-90.632,-93.958,166.013,50.249,159.046
C01408=1021.291,-90.881,-93.948,166.010,50.253,159.046
C01409=1021.285,-91.131,-93.938,166.007,50.258,159.046
C01410=1021.280,-91.381,-93.929,166.004,50.261,159.046
C01411=1021.274,-91.631,-93.920,166.001,50.265,159.047
C01412=1021.269,-91.880,-93.911,165.998,50.269,159.047
C01413=1021.263,-92.130,-93.900,165.995,50.274,159.047
C01414=1021.257,-92.380,-93.891,165.991,50.277,159.047
C01415=1021.253,-92.630,-93.882,165.989,50.281,159.047
C01416=1021.246,-92.880,-93.872,165.986,50.285,159.048
C01417=1021.242,-93.129,-93.862,165.982,50.290,159.048
C01418=1021.235,-93.379,-93.853,165.979,50.293,159.048
C01419=1021.231,-93.629,-93.844,165.977,50.297,159.048
C01420=1021.225,-93.879,-93.834,165.974,50.301,159.048
C01421=1021.219,-94.128,-93.825,165.970,50.305,159.048
C01422=1021.214,-94.378,-93.816,165.967,50.309,159.049
C01423=1021.208,-94.627,-93.806,165.964,50.313,159.049
C01424=1021.203,-94.878,-93.796,165.962,50.317,159.049
C01425=1021.197,-95.127,-93.787,165.958,50.321,159.049
C01426=1021.192,-95.377,-93.778,165.955,50.325,159.049
C01427=1021.187,-95.627,-93.768,165.952,50.329,159.050
C01428=1021.181,-95.876,-93.759,165.949,50.333,159.050
C01429=1021.176,-96.126,-93.750,165.945,50.337,159.050
C01430=1021.170,-96.375,-93.741,165.943,50.341,159.050
C01431=1021.165,-96.626,-93.731,165.940,50.345,159.050
C01432=1021.160,-96.875,-93.722,165.937,50.349,159.051
C01433=1021.154,-97.125,-93.712,165.933,50.353,159.051
C01434=1021.149,-97.375,-93.703,165.930,50.357,159.051
C01435=1021.143,-97.625,-93.694,165.927,50.361,159.051
C01436=1021.138,-97.875,-93.685,165.925,50.365,159.051
C01437=1021.133,-98.124,-93.675,165.921,50.369,159.051
C01438=1021.127,-98.374,-93.667,165.918,50.373,159.052
C01439=1021.121,-98.624,-93.657,165.915,50.377,159.052
C01440=1021.115,-98.874,-93.649,165.912,50.381,159.052
C01441=1021.111,-99.123,-93.639,165.909,50.385,159.052
C01442=1021.105,-99.374,-93.630,165.906,50.389,159.052
C01443=1021.099,-99.623,-93.621,165.904,50.394,159.053
C01444=1021.094,-99.873,-93.612,165.900,50.398,159.053
C01445=1021.088,-100.123,-93.603,165.897,50.401,159.053
C01446=1021.082,-100.372,-93.594,165.894,50.405,159.053
C01447=1021.077,-100.622,-93.586,165.890,50.410,159.053
C01448=1021.072,-100.872,-93.575,165.888,50.414,159.054
C01449=1021.066,-101.157,-93.566,165.884,50.418,159.054
C01450=1021.059,-101.441,-93.556,165.881,50.424,159.054
C01451=1021.053,-101.726,-93.546,165.877,50.428,159.054
C01452=1021.047,-102.010,-93.535,165.873,50.432,159.054
C01453=1021.041,-102.261,-93.526,165.870,50.437,159.055
C01454=1021.035,-102.510,-93.517,165.868,50.441,159.055
C01455=1021.030,-102.760,-93.509,165.865,50.445,159.055
C01456=1021.024,-103.010,-93.500,165.861,50.449,159.055
C01457=1021.019,-103.260,-93.490,165.858,50.453,159.055
C01458=1021.014,-103.509,-93.482,165.856,50.457,159.056
C01459=1021.008,-103.760,-93.473,165.852,50.461,159.056
C01460=1021.003,-104.009,-93.464,165.849,50.465,159.056
C01461=1020.998,-104.258,-93.455,165.846,50.469,159.056
C01462=1020.992,-104.508,-93.447,165.842,50.473,159.056
C01463=1020.986,-104.759,-93.438,165.840,50.477,159.057
C01464=1020.981,-105.008,-93.429,165.837,50.481,159.057
C01465=1020.976,-105.257,-93.420,165.834,50.486,159.057
C01466=1020.971,-105.507,-93.411,165.830,50.489,159.057
C01467=1020.965,-105.758,-93.402,165.828,50.493,159.057
C01468=1020.960,-106.008,-93.394,165.825,50.497,159.058
C01469=1020.955,-106.257,-93.385,165.822,50.502,159.058
C01470=1020.949,-106.506,-93.376,165.818,50.506,159.058
C01471=1020.943,-106.757,-93.367,165.815,50.509,159.058
C01472=1020.938,-107.007,-93.359,165.813,50.514,159.058
C01473=1020.933,-107.256,-93.350,165.809,50.518,159.058
C01474=1020.927,-107.506,-93.342,165.806,50.522,159.059
C01475=1020.922,-107.756,-93.333,165.803,50.526,159.059
C01476=1020.916,-108.006,-93.324,165.800,50.530,159.059
C01477=1020.911,-108.255,-93.315,165.797,50.534,159.059
C01478=1020.905,-108.505,-93.307,165.794,50.538,159.059
C01479=1020.900,-108.755,-93.298,165.791,50.542,159.060
C01480=1020.894,-109.005,-93.289,165.788,50.547,159.060
C01481=1020.889,-109.255,-93.281,165.785,50.551,159.060
C01482=1020.884,-109.504,-93.272,165.782,50.554,159.060
C01483=1020.879,-109.754,-93.264,165.778,50.559,159.060
C01484=1020.873,-110.004,-93.256,165.776,50.563,159.060
C01485=1020.867,-110.253,-93.247,165.773,50.567,159.061
C01486=1020.861,-110.504,-93.239,165.769,50.572,159.061
C01487=1020.856,-110.753,-93.230,165.767,50.576,159.061
C01488=1020.851,-111.003,-93.222,165.764,50.579,159.061
C01489=1020.846,-111.253,-93.213,165.760,50.584,159.061
C01490=1020.840,-111.503,-93.205,165.757,50.588,159.062
C01491=1020.835,-111.752,-93.196,165.754,50.592,159.062
C01492=1020.830,-112.002,-93.188,165.752,50.596,159.062
C01493=1020.825,-112.252,-93.179,165.748,50.600,159.062
C01494=1020.819,-112.501,-93.171,165.745,50.604,159.062
C01495=1020.813,-112.752,-93.162,165.742,50.608,159.063
C01496=1020.808,-113.002,-93.155,165.739,50.612,159.063
C01497=1020.802,-113.252,-93.146,165.736,50.617,159.063
C01498=1020.797,-113.501,-93.138,165.733,50.620,159.063
C01499=1020.792,-113.751,-93.129,165.729,50.624,159.063
C01500=1020.787,-114.001,-93.121,165.726,50.629,159.063
C01501=1020.781,-114.250,-93.112,165.724,50.633,159.064
C01502=1020.776,-114.500,-93.104,165.721,50.637,159.064
C01503=1020.771,-114.750,-93.095,165.717,50.641,159.064
C01504=1020.765,-115.000,-93.088,165.714,50.645,159.064
C01505=1020.760,-115.250,-93.080,165.712,50.649,159.064
C01506=1020.755,-115.499,-93.071,165.708,50.653,159.064
C01507=1020.749,-115.749,-93.063,165.705,50.657,159.065
C01508=1020.743,-115.998,-93.055,165.703,50.662,159.065
C01509=1020.738,-116.249,-93.047,165.699,50.665,159.065
C01510=1020.733,-116.499,-93.039,165.696,50.669,159.065
C01511=1020.728,-116.748,-93.030,165.693,50.674,159.065
C01512=1020.723,-116.998,-93.022,165.690,50.678,159.066
C01513=1020.716,-117.282,-93.013,165.687,50.682,159.066
C01514=1020.709,-117.567,-93.003,165.683,50.687,159.066
C01515=1020.704,-117.852,-92.994,165.680,50.692,159.066
C01516=1020.698,-118.137,-92.985,165.676,50.696,159.066
C01517=1020.693,-118.387,-92.977,165.673,50.700,159.067
C01518=1020.687,-118.636,-92.969,165.670,50.705,159.067
C01519=1020.682,-118.886,-92.961,165.667,50.709,159.067
C01520=1020.676,-119.136,-92.952,165.664,50.713,159.067
C01521=1020.671,-119.386,-92.944,165.660,50.717,159.067
C01522=1020.665,-119.636,-92.937,165.658,50.721,159.067
C01523=1020.660,-119.886,-92.928,165.655,50.725,159.068
C01524=1020.655,-120.135,-92.920,165.652,50.729,159.068
C01525=1020.650,-120.385,-92.913,165.648,50.734,159.068
C01526=1020.644,-120.634,-92.905,165.646,50.738,159.068
C01527=1020.639,-120.884,-92.896,165.643,50.741,159.068
C01528=1020.634,-121.134,-92.888,165.639,50.746,159.068
C01529=1020.628,-121.384,-92.880,165.636,50.750,159.069
C01530=1020.623,-121.634,-92.873,165.634,50.754,159.069
C01531=1020.618,-121.884,-92.864,165.631,50.758,159.069
C01532=1020.612,-122.134,-92.857,165.627,50.762,159.069
C01533=1020.607,-122.384,-92.848,165.624,50.766,159.069
C01534=1020.603,-122.633,-92.841,165.622,50.770,159.070
C01535=1020.597,-122.883,-92.833,165.618,50.775,159.070
C01536=1020.592,-123.133,-92.825,165.615,50.779,159.070
C01537=1020.586,-123.383,-92.817,165.612,50.782,159.070
C01538=1020.581,-123.633,-92.810,165.610,50.787,159.070
C01539=1020.575,-123.882,-92.801,165.606,50.791,159.070
C01540=1020.570,-124.132,-92.794,165.603,50.795,159.071
C01541=1020.565,-124.381,-92.786,165.600,50.799,159.071
C01542=1020.560,-124.632,-92.778,165.596,50.803,159.071
C01543=1020.554,-124.881,-92.770,165.594,50.807,159.071
C01544=1020.549,-125.132,-92.763,165.591,50.812,159.071
C01545=1020.543,-125.381,-92.755,165.588,50.816,159.072
C01546=1020.538,-125.631,-92.747,165.585,50.820,159.072
C01547=1020.533,-125.881,-92.740,165.582,50.824,159.072
C01548=1020.528,-126.130,-92.732,165.579,50.828,159.072
C01549=1020.522,-126.380,-92.724,165.575,50.832,159.072
C01550=1020.517,-126.631,-92.717,165.573,50.836,159.072
C01551=1020.512,-126.880,-92.708,165.570,50.841,159.073
C01552=1020.507,-127.130,-92.701,165.566,50.845,159.073
C01553=1020.502,-127.380,-92.694,165.564,50.849,159.073
C01554=1020.496,-127.629,-92.686,165.561,50.853,159.073
C01555=1020.491,-127.879,-92.679,165.558,50.857,159.073
C01556=1020.486,-128.129,-92.670,165.554,50.861,159.073
C01557=1020.481,-128.378,-92.662,165.551,50.865,159.074
C01558=1020.476,-128.628,-92.653,165.549,50.868,159.074
C01559=1020.473,-128.877,-92.644,165.546,50.871,159.074
C01560=1020.469,-129.127,-92.633,165.543,50.872,159.073
C01561=1020.467,-129.377,-92.624,165.540,50.874,159.073
C01562=1020.464,-129.626,-92.612,165.538,50.875,159.073
C01563=1020.462,-129.877,-92.599,165.536,50.875,159.073
C01564=1020.461,-130.126,-92.587,165.534,50.875,159.072
C01565=1020.460,-130.376,-92.575,165.531,50.874,159.072
C01566=1020.459,-130.625,-92.561,165.529,50.873,159.071
C01567=1020.460,-130.875,-92.546,165.527,50.871,159.070
C01568=1020.459,-131.125,-92.532,165.524,50.869,159.070
C01569=1020.460,-131.375,-92.516,165.522,50.867,159.069
C01570=1020.461,-131.625,-92.501,165.520,50.864,159.068
C01571=1020.464,-131.874,-92.484,165.519,50.860,159.067
C01572=1020.466,-132.124,-92.467,165.516,50.856,159.066
C01573=1020.469,-132.374,-92.449,165.515,50.851,159.065
C01574=1020.472,-132.623,-92.431,165.513,50.846,159.064
C01575=1020.475,-132.874,-92.413,165.512,50.840,159.063
C01576=1020.480,-133.123,-92.392,165.510,50.834,159.061
C01577=1020.202,-133.149,-92.753,165.465,51.144,159.106
C01578=1020.198,-132.900,-92.772,165.466,51.150,159.107
C01579=1020.194,-132.650,-92.792,165.468,51.156,159.108
C01580=1020.191,-132.400,-92.809,165.470,51.161,159.110
C01581=1020.188,-132.150,-92.828,165.472,51.165,159.111
C01582=1020.186,-131.900,-92.844,165.473,51.170,159.112
C01583=1020.184,-131.651,-92.861,165.475,51.174,159.113
C01584=1020.182,-131.401,-92.877,165.478,51.176,159.114
C01585=1020.182,-131.151,-92.892,165.479,51.179,159.115
C01586=1020.182,-130.902,-92.907,165.481,51.181,159.115
C01587=1020.182,-130.652,-92.921,165.484,51.183,159.116
C01588=1020.182,-130.402,-92.935,165.485,51.184,159.116
C01589=1020.183,-130.152,-92.948,165.488,51.185,159.117
C01590=1020.184,-129.903,-92.960,165.491,51.185,159.118
C01591=1020.186,-129.652,-92.973,165.493,51.184,159.118
C01592=1020.189,-129.403,-92.983,165.496,51.183,159.118
C01593=1020.192,-129.153,-92.994,165.499,51.182,159.118
C01594=1020.195,-128.903,-93.005,165.502,51.180,159.119
C01595=1020.198,-128.654,-93.014,165.504,51.178,159.119
C01596=1020.202,-128.404,-93.023,165.507,51.174,159.119
C01597=1020.207,-128.155,-93.031,165.510,51.171,159.119
C01598=1020.212,-127.905,-93.039,165.513,51.167,159.119
C01599=1020.218,-127.656,-93.047,165.516,51.163,159.118
C01600=1020.223,-127.405,-93.054,165.518,51.159,159.118
C01601=1020.228,-127.157,-93.062,165.522,51.154,159.118
C01602=1020.233,-126.906,-93.070,165.525,51.150,159.118
C01603=1020.239,-126.656,-93.077,165.527,51.146,159.117
C01604=1020.244,-126.407,-93.085,165.531,51.141,159.117
C01605=1020.249,-126.157,-93.092,165.534,51.137,159.117
C01606=1020.254,-125.907,-93.100,165.536,51.133,159.117
C01607=1020.260,-125.658,-93.108,165.540,51.129,159.117
C01608=1020.265,-125.407,-93.115,165.543,51.125,159.117
C01609=1020.270,-125.158,-93.122,165.547,51.121,159.117
C01610=1020.275,-124.908,-93.131,165.549,51.116,159.116
C01611=1020.281,-124.658,-93.138,165.552,51.112,159.116
C01612=1020.286,-124.408,-93.146,165.556,51.108,159.116
C01613=1020.291,-124.158,-93.154,165.558,51.103,159.116
C01614=1020.297,-123.908,-93.161,165.561,51.099,159.115
C01615=1020.302,-123.659,-93.170,165.564,51.096,159.115
C01616=1020.307,-123.409,-93.177,165.568,51.091,159.115
C01617=1020.313,-123.159,-93.185,165.570,51.087,159.115
C01618=1020.318,-122.909,-93.193,165.573,51.083,159.115
C01619=1020.323,-122.659,-93.201,165.576,51.078,159.115
C01620=1020.329,-122.409,-93.209,165.579,51.074,159.114
C01621=1020.333,-122.160,-93.217,165.582,51.071,159.114
C01622=1020.338,-121.910,-93.224,165.586,51.066,159.114
C01623=1020.344,-121.660,-93.232,165.588,51.062,159.114
C01624=1020.349,-121.410,-93.240,165.591,51.058,159.114
C01625=1020.354,-121.160,-93.249,165.595,51.053,159.114
C01626=1020.360,-120.910,-93.256,165.597,51.049,159.113
C01627=1020.365,-120.661,-93.264,165.600,51.046,159.113
C01628=1020.370,-120.410,-93.272,165.604,51.041,159.113
C01629=1020.376,-120.161,-93.280,165.607,51.037,159.113
C01630=1020.381,-119.912,-93.288,165.609,51.033,159.113
C01631=1020.386,-119.662,-93.296,165.613,51.028,159.113
C01632=1020.392,-119.412,-93.304,165.616,51.024,159.112
C01633=1020.397,-119.163,-93.312,165.618,51.020,159.112
C01634=1020.402,-118.912,-93.320,165.622,51.016,159.112
C01635=1020.407,-118.662,-93.328,165.625,51.012,159.112
C01636=1020.413,-118.412,-93.336,165.628,51.008,159.112
C01637=1020.418,-118.163,-93.344,165.631,51.004,159.111
C01638=1020.424,-117.879,-93.353,165.635,50.998,159.111
C01639=1020.430,-117.594,-93.363,165.638,50.994,159.111
C01640=1020.437,-117.310,-93.371,165.641,50.990,159.111
C01641=1020.443,-117.025,-93.381,165.644,50.984,159.110
C01642=1020.448,-116.775,-93.389,165.648,50.980,159.110
C01643=1020.453,-116.525,-93.397,165.651,50.976,159.110
C01644=1020.458,-116.275,-93.406,165.654,50.972,159.110
C01645=1020.464,-116.026,-93.414,165.657,50.968,159.110
C01646=1020.470,-115.776,-93.422,165.660,50.964,159.110
C01647=1020.475,-115.526,-93.430,165.663,50.959,159.109
C01648=1020.480,-115.276,-93.438,165.666,50.955,159.109
C01649=1020.485,-115.026,-93.447,165.669,50.951,159.109
C01650=1020.491,-114.777,-93.455,165.673,50.946,159.109
C01651=1020.496,-114.527,-93.462,165.675,50.942,159.109
C01652=1020.501,-114.277,-93.471,165.678,50.939,159.109
C01653=1020.507,-114.027,-93.479,165.682,50.934,159.108
C01654=1020.512,-113.777,-93.488,165.685,50.930,159.108
C01655=1020.517,-113.528,-93.496,165.687,50.926,159.108
C01656=1020.522,-113.278,-93.505,165.690,50.922,159.108
C01657=1020.528,-113.028,-93.513,165.694,50.918,159.108
C01658=1020.534,-112.779,-93.521,165.697,50.914,159.108
C01659=1020.539,-112.529,-93.529,165.699,50.910,159.107
C01660=1020.545,-112.278,-93.538,165.703,50.905,159.107
C01661=1020.550,-112.028,-93.546,165.706,50.901,159.107
C01662=1020.555,-111.779,-93.555,165.708,50.897,159.107
C01663=1020.560,-111.529,-93.563,165.712,50.892,159.106
C01664=1020.566,-111.279,-93.572,165.715,50.889,159.106
C01665=1020.571,-111.030,-93.580,165.718,50.885,159.106
C01666=1020.576,-110.780,-93.589,165.722,50.880,159.106
C01667=1020.581,-110.530,-93.597,165.724,50.876,159.106
C01668=1020.587,-110.281,-93.605,165.728,50.872,159.106
C01669=1020.593,-110.030,-93.614,165.731,50.867,159.105
C01670=1020.599,-109.781,-93.623,165.733,50.863,159.105
C01671=1020.604,-109.531,-93.631,165.737,50.859,159.105
C01672=1020.609,-109.281,-93.639,165.740,50.855,159.105
C01673=1020.614,-109.031,-93.648,165.743,50.851,159.105
C01674=1020.620,-108.782,-93.656,165.746,50.847,159.105
C01675=1020.625,-108.532,-93.665,165.749,50.843,159.104
C01676=1020.631,-108.282,-93.674,165.752,50.838,159.104
C01677=1020.636,-108.032,-93.682,165.755,50.834,159.104
C01678=1020.641,-107.782,-93.691,165.758,50.830,159.104
C01679=1020.647,-107.532,-93.699,165.761,50.826,159.103
C01680=1020.652,-107.283,-93.708,165.764,50.821,159.103
C01681=1020.658,-107.032,-93.717,165.767,50.818,159.103
C01682=1020.663,-106.783,-93.725,165.770,50.814,159.103
C01683=1020.668,-106.533,-93.734,165.774,50.809,159.103
C01684=1020.674,-106.284,-93.743,165.776,50.805,159.103
C01685=1020.679,-106.034,-93.751,165.779,50.801,159.102
C01686=1020.685,-105.784,-93.760,165.783,50.796,159.102
C01687=1020.690,-105.534,-93.769,165.786,50.793,159.102
C01688=1020.695,-105.284,-93.777,165.788,50.789,159.102
C01689=1020.701,-105.035,-93.786,165.792,50.784,159.102
C01690=1020.707,-104.785,-93.795,165.795,50.780,159.101
C01691=1020.711,-104.535,-93.804,165.797,50.776,159.101
C01692=1020.717,-104.285,-93.813,165.801,50.772,159.101
C01693=1020.722,-104.036,-93.822,165.804,50.768,159.101
C01694=1020.728,-103.785,-93.831,165.807,50.764,159.101
C01695=1020.733,-103.536,-93.839,165.810,50.759,159.101
C01696=1020.739,-103.286,-93.848,165.813,50.755,159.100
C01697=1020.744,-103.037,-93.857,165.816,50.751,159.100
C01698=1020.750,-102.786,-93.866,165.819,50.747,159.100
C01699=1020.755,-102.536,-93.875,165.823,50.743,159.100
C01700=1020.760,-102.287,-93.884,165.825,50.739,159.100
C01701=1020.766,-102.037,-93.893,165.829,50.735,159.099
C01702=1020.772,-101.752,-93.902,165.832,50.730,159.099
C01703=1020.779,-101.468,-93.913,165.835,50.725,159.099
C01704=1020.785,-101.183,-93.924,165.839,50.721,159.099
C01705=1020.791,-100.898,-93.933,165.842,50.716,159.098
C01706=1020.796,-100.649,-93.942,165.846,50.711,159.098
C01707=1020.802,-100.400,-93.951,165.848,50.707,159.098
C01708=1020.808,-100.149,-93.960,165.851,50.704,159.098
C01709=1020.812,-99.900,-93.969,165.855,50.699,159.098
C01710=1020.818,-99.650,-93.978,165.858,50.695,159.098
C01711=1020.824,-99.400,-93.987,165.860,50.691,159.097
C01712=1020.829,-99.151,-93.996,165.864,50.687,159.097
C01713=1020.835,-98.900,-94.005,165.867,50.682,159.097
C01714=1020.841,-98.651,-94.014,165.870,50.678,159.097
C01715=1020.846,-98.401,-94.022,165.873,50.674,159.096
C01716=1020.851,-98.151,-94.033,165.876,50.670,159.096
C01717=1020.857,-97.901,-94.041,165.879,50.665,159.096
C01718=1020.863,-97.652,-94.051,165.882,50.662,159.096
C01719=1020.867,-97.402,-94.060,165.885,50.658,159.096
C01720=1020.873,-97.152,-94.069,165.888,50.653,159.095
C01721=1020.879,-96.902,-94.078,165.892,50.649,159.095
C01722=1020.883,-96.653,-94.088,165.895,50.646,159.095
C01723=1020.889,-96.402,-94.096,165.897,50.641,159.095
C01724=1020.894,-96.153,-94.106,165.901,50.637,159.095
C01725=1020.900,-95.903,-94.116,165.904,50.633,159.095
C01726=1020.905,-95.653,-94.125,165.907,50.629,159.094
C01727=1020.911,-95.403,-94.134,165.909,50.625,159.094
C01728=1020.917,-95.154,-94.144,165.913,50.621,159.094
C01729=1020.921,-94.904,-94.153,165.916,50.617,159.094
C01730=1020.927,-94.654,-94.162,165.919,50.613,159.094
C01731=1020.932,-94.405,-94.172,165.922,50.609,159.094
C01732=1020.938,-94.155,-94.181,165.925,50.605,159.093
C01733=1020.944,-93.905,-94.190,165.928,50.601,159.093
C01734=1020.949,-93.655,-94.200,165.931,50.597,159.093
C01735=1020.954,-93.406,-94.209,165.934,50.593,159.093
C01736=1020.960,-93.156,-94.219,165.937,50.589,159.093
C01737=1020.965,-92.906,-94.228,165.940,50.585,159.092
C01738=1020.970,-92.656,-94.238,165.944,50.580,159.092
C01739=1020.976,-92.407,-94.247,165.947,50.577,159.092
C01740=1020.981,-92.156,-94.257,165.949,50.573,159.092
C01741=1020.987,-91.907,-94.266,165.952,50.568,159.092
C01742=1020.993,-91.657,-94.275,165.956,50.564,159.091
C01743=1020.998,-91.408,-94.285,165.958,50.560,159.091
C01744=1021.004,-91.158,-94.294,165.961,50.556,159.091
C01745=1021.009,-90.908,-94.304,165.965,50.552,159.091
C01746=1021.015,-90.659,-94.314,165.968,50.548,159.091
C01747=1021.019,-90.409,-94.323,165.970,50.544,159.090
C01748=1021.026,-90.159,-94.332,165.974,50.539,159.090
C01749=1021.031,-89.909,-94.343,165.977,50.535,159.090
C01750=1021.037,-89.660,-94.352,165.979,50.531,159.090
C01751=1021.043,-89.410,-94.361,165.984,50.527,159.090
C01752=1021.047,-89.160,-94.370,165.986,50.523,159.089
C01753=1021.053,-88.910,-94.380,165.989,50.519,159.089
C01754=1021.059,-88.660,-94.390,165.993,50.515,159.089
C01755=1021.064,-88.411,-94.399,165.995,50.511,159.089
C01756=1021.070,-88.161,-94.410,165.998,50.506,159.089
C01757=1021.075,-87.912,-94.419,166.002,50.502,159.088
C01758=1021.081,-87.661,-94.429,166.004,50.498,159.088
C01759=1021.087,-87.412,-94.438,166.007,50.494,159.088
C01760=1021.092,-87.162,-94.448,166.011,50.490,159.088
C01761=1021.098,-86.912,-94.457,166.014,50.486,159.088
C01762=1021.104,-86.662,-94.467,166.016,50.482,159.087
C01763=1021.109,-86.413,-94.476,166.020,50.477,159.087
C01764=1021.115,-86.163,-94.486,166.023,50.473,159.087
C01765=1021.120,-85.913,-94.496,166.025,50.469,159.087
C01766=1021.126,-85.631,-94.507,166.029,50.465,159.086
C01767=1021.133,-85.348,-94.518,166.033,50.460,159.086
C01768=1021.139,-85.066,-94.529,166.036,50.455,159.086
C01769=1021.145,-84.783,-94.540,166.040,50.450,159.086
C01770=1021.152,-84.533,-94.549,166.042,50.446,159.085
C01771=1021.156,-84.284,-94.559,166.046,50.442,159.085
C01772=1021.163,-84.034,-94.569,166.049,50.438,159.085
C01773=1021.168,-83.784,-94.579,166.052,50.434,159.085
C01774=1021.174,-83.534,-94.588,166.055,50.430,159.085
C01775=1021.179,-83.285,-94.598,166.058,50.425,159.084
C01776=1021.185,-83.035,-94.608,166.061,50.421,159.084
C01777=1021.191,-82.785,-94.618,166.064,50.417,159.084
C01778=1021.197,-82.535,-94.627,166.067,50.413,159.084
C01779=1021.202,-82.286,-94.638,166.070,50.409,159.083
C01780=1021.208,-82.036,-94.648,166.074,50.404,159.083
C01781=1021.214,-81.786,-94.658,166.076,50.400,159.083
C01782=1021.220,-81.536,-94.667,166.079,50.396,159.083
C01783=1021.225,-81.287,-94.677,166.083,50.392,159.083
C01784=1021.231,-81.037,-94.687,166.085,50.387,159.082
C01785=1021.236,-80.787,-94.697,166.089,50.383,159.082
C01786=1021.242,-80.537,-94.706,166.092,50.379,159.082
C01787=1021.247,-80.288,-94.716,166.094,50.375,159.082
C01788=1021.253,-80.038,-94.726,166.098,50.370,159.081
C01789=1021.259,-79.789,-94.737,166.101,50.366,159.081
C01790=1021.265,-79.539,-94.747,166.103,50.362,159.081
C01791=1021.270,-79.288,-94.757,166.107,50.359,159.081
C01792=1021.276,-79.039,-94.766,166.110,50.354,159.081
C01793=1021.281,-78.790,-94.777,166.113,50.350,159.080
C01794=1021.287,-78.540,-94.787,166.116,50.346,159.080
C01795=1021.292,-78.290,-94.797,166.119,50.342,159.080
